// TIA Portal project "04_Kommisionierung_2018-10-11" (V14)
// Automatikbetribeb für das Modul "04-Kommisionierung" mit Factory IO

(* hardware
DEVICE "S7300/ET200M-Station_4"  S7-300 station
   slot 0: "Profilschiene_0"  Rail  6ES7 390-1***0-0AA0
   slot 1: "PS 307 5A_1"  PS 307 5A  6ES7 307-1EA01-0AA0
   slot 2: "PLC_Bus"  CPU 314C-2 DP  6ES7 314-6CH04-0AB0  V3.3
      slot 0: "MPI-Schnittstelle_1"  MPI
      slot 1: "DP-Schnittstelle_1"  DP
      slot 2: "DI 24/DO 16_1"  DI24/DO16
      slot 3: "AI 5/AO 2_1"  AI5/AO2
      slot 4: "Zählen_1"  Counter
      slot 5: "Positionieren_1"  Positioning
   slot 4: "DI 64x24VDC sinking/souring_1"  DI64 x 24VDC  6ES7 321-1BP00-0AA0
   slot 5: "DI 64x24VDC sinking/souring_2"  DI64 x 24VDC  6ES7 321-1BP00-0AA0
   slot 6: "DI 64x24VDC sinking/souring_3"  DI64 x 24VDC  6ES7 321-1BP00-0AA0
   slot 7: "DI 64x24VDC sinking/souring_4"  DI64 x 24VDC  6ES7 321-1BP00-0AA0
   slot 8: "DO 64x24VDC/0.3A sourcing_1"  DO64 x 24VDC / 0.3A, P  6ES7 322-1BP00-0AA0
   slot 9: "DO 64x24VDC/0.3A sourcing_2"  DO64 x 24VDC / 0.3A, P  6ES7 322-1BP00-0AA0
   slot 10: "DO 64x24VDC/0.3A sourcing_3"  DO64 x 24VDC / 0.3A, P  6ES7 322-1BP00-0AA0
   slot 11: "DO 64x24VDC/0.3A sourcing_4"  DO64 x 24VDC / 0.3A, P  6ES7 322-1BP00-0AA0
*)

// ===== PLC "PLC_Bus"  CPU 314C-2 DP =====

VAR_GLOBAL   // PLC tag table "Betriebsart"
   "S0_HS" AT %E0.0 : Bool;   // Hauptschalter 0-Aus, 1-Ein
   "S1_Not_Halt" AT %E0.1 : Bool;   // Not-Halt NC
   "S2_START" AT %E0.2 : Bool;   // Taster START NO
   "S3_STOP" AT %E0.3 : Bool;   // Taster STOP NC
   "Res_E04" AT %E0.4 : Bool;
   "Res_E05" AT %E0.5 : Bool;
   "Res_E06" AT %E0.6 : Bool;
   "Res_E07" AT %E0.7 : Bool;
   "Res_E10" AT %E1.0 : Bool;
   "Res_E11" AT %E1.1 : Bool;
   "Res_E12" AT %E1.2 : Bool;
   "Res_E13" AT %E1.3 : Bool;
   "Res_E14" AT %E1.4 : Bool;
   "Res_E15" AT %E1.5 : Bool;
   "Res_E16" AT %E1.6 : Bool;
   "Factory_IO_RUN" AT %E1.7 : Bool;   // Rückmeldung Factory IO läuft
   "P1_MS_RT" AT %A1.0 : Bool;   // Meldesäule Rot
   "P2_MS_GE" AT %A0.1 : Bool;   // Meldesäule Gelb
   "P3_MS_GN" AT %A0.2 : Bool;   // Meldesäule Grün
   "P10_START" AT %A0.3 : Bool;   // Anzeige grün in START-Taster
   "P11_STOP" AT %A0.4 : Bool;   // Anzeige gelb in STOP-Taster
   "Res_A0.5" AT %A0.5 : Bool;
   "P12_Anfahrwarnung" AT %A0.6 : Bool;   // Rundumleuchte System
   "P13_Sirene" AT %A0.7 : Bool;   // Sirene System
   "Res_A10" AT %A1.0 : Bool;
   "Res_A11" AT %A1.1 : Bool;
   "Res_A12" AT %A1.2 : Bool;
   "Res_A13" AT %A1.3 : Bool;
   "Res_A14" AT %A1.4 : Bool;
   "Res_A15" AT %A1.5 : Bool;
   "Res_A16" AT %A1.6 : Bool;
   "Res_A17" AT %A1.7 : Bool;
   "Log_1" AT %M0.1 : Bool;   // statisch "1"
   "Log_0" AT %M0.0 : Bool;   // statisch "0"
   "Takt_1HZ" AT %M100.5 : Bool;   // Taktmerker 1 Hz
END_VAR

VAR_GLOBAL   // PLC tag table "Kommisionierung"
   "B5001_TB5001" AT %E10.0 : Bool;   // Teil vom Emiiter vorhanden
   "B5002_TB5001" AT %E10.1 : Bool;   // Transportband-Ende
   "B5003_TB5002" AT %E10.2 : Bool;   // Transportband-Anfang
   "B5004_TB5002" AT %E10.3 : Bool;   // Transportband-Ende
   "B5005_TB5003" AT %E10.4 : Bool;   // Transportband-Anfang
   "B5006_TB5003" AT %E10.5 : Bool;   // Transportband-Ende
   "B5007_TB5004" AT %E10.6 : Bool;   // Transportband-Anfang
   "B5008_TB5004" AT %E10.7 : Bool;   // Transportband-Ende
   "B5009_TB5005" AT %E11.0 : Bool;   // Transportband-Anfang
   "B5010_TB5005" AT %E11.1 : Bool;   // Transportband-Ende
   "B5011_Farbteil_BL" AT %E11.2 : Bool;   // Farberkennung BL
   "B5012_Farbteil_GN" AT %E11.3 : Bool;   // Farberkennung GN
   "B5013_TB5006" AT %E11.4 : Bool;   // Transportband-Anfang
   "B5014_TB5006" AT %E11.5 : Bool;   // Transportband-Ende
   "B5015_Teil_in_Pos" AT %E11.6 : Bool;   // Teil in Abholposition
   "B5016_Teil_vorhanden" AT %E11.7 : Bool;   // Teil vom Emitter generiert
   "B5017_Teil_in_Pos" AT %E12.0 : Bool;   // Teil in Abholposition
   "B5018_Teil_vorhanden" AT %E12.1 : Bool;   // Teil vom Emitter generiert
   "B5019_TB5009" AT %E12.2 : Bool;   // Transportband-Anfang
   "B5020_TB5009" AT %E12.3 : Bool;   // Transportband-Ende
   "B5021_TB5010" AT %E12.4 : Bool;   // Transportband-Anfang
   "B5022_TB5010" AT %E12.5 : Bool;   // Transportband-Ende
   "Res_E126" AT %E12.6 : Bool;
   "Res_E127" AT %E12.7 : Bool;
   "B5030_PAP5001_RM_X" AT %E13.0 : Bool;
   "B5031_PAP5001_RM_Z" AT %E13.1 : Bool;
   "B5032_PAP5001_Teil_erkannt" AT %E13.2 : Bool;
   "B5040_PAP5002_RM_X" AT %E13.3 : Bool;
   "B5041_PAP5002_RM_Z" AT %E13.4 : Bool;
   "B5042_PAP5002_Teil_erkannt" AT %E13.5 : Bool;
   "Res_E136" AT %E13.6 : Bool;
   "Res_E137" AT %E13.7 : Bool;
   "TB5001" AT %A8.0 : Bool;
   "TB5002" AT %A8.1 : Bool;
   "TB5003" AT %A8.2 : Bool;
   "TB5004" AT %A8.3 : Bool;
   "TB5005" AT %A8.4 : Bool;
   "TB5006" AT %A8.5 : Bool;
   "TB5007" AT %A8.6 : Bool;
   "TB5008" AT %A8.7 : Bool;
   "TB5009" AT %A9.0 : Bool;
   "TB5010" AT %A9.1 : Bool;
   "STOP5001" AT %A9.2 : Bool;   // Stopper
   "STOP5002" AT %A9.3 : Bool;   // Stopper
   "STOP5003" AT %A9.4 : Bool;   // Stopper
   "STOP5004" AT %A9.5 : Bool;   // Stopper
   "STOP5005" AT %A9.6 : Bool;   // Stopper
   "Res_A97" AT %A9.7 : Bool;
   "PAP5001_X" AT %A10.0 : Bool;
   "PAP5001_Z" AT %A10.1 : Bool;
   "PAP5001_Greifer" AT %A10.2 : Bool;
   "PAP5002_X" AT %A10.3 : Bool;
   "PAP5002_Z" AT %A10.4 : Bool;
   "PAP5002_Greifer" AT %A10.5 : Bool;
   "Res_A106" AT %A10.6 : Bool;
   "Res_A107" AT %A10.7 : Bool;
   "RS5001_V" AT %A11.0 : Bool;   // Rollensorter Antrieb ein
   "RS5001_links" AT %A11.1 : Bool;   // Rollensorter Steuerung links
   "RS5001_rechts" AT %A11.2 : Bool;   // Rollensorter Steuerung rechts
   "Res_A113" AT %A11.3 : Bool;
   "Res_A114" AT %A11.4 : Bool;
   "Emitter_1" AT %A11.5 : Bool;
   "Emitter_2" AT %A11.6 : Bool;
   "Emitter_3" AT %A11.7 : Bool;
END_VAR

VAR_GLOBAL   // PLC tag table "KW_Variablen"
   "M_True" AT %M20.0 : Bool;   // Merker, der immer TRUE ist
   "M_False" AT %M20.1 : Bool;   // Merker, der immer FALSE ist
   "M_Beladen_Fern" AT %M22.0 : Bool;   // Merker, das Signal die ferne Ladestation zu aktivieren
   "M_Beladen_Nah" AT %M22.1 : Bool;   // Merker, das Signal die nähe Ladestation zu aktivieren
   "M_Abfuhr_Fern" AT %M22.2 : Bool;   // Merker, das Signal, dass das laden bei der fernen Ladestation beendet ist
   "M_Abfuhr_Nah" AT %M22.3 : Bool;   // Merker, das Signal, dass das laden bei der nähren Ladestation beendet ist
   "M_FRG_N1" AT %M22.4 : Bool;   // Merker, Freigabe Nummer 1
   "M_BND2_KB" AT %M22.5 : Bool;   // Merker Kiste beladen für das zweite Band
   "M_BND3_KB" AT %M22.6 : Bool;   // Merker Kiste beladen für das dritte Band
   "M_BND4_KB" AT %M22.7 : Bool;   // Merker Kiste beladen für das vierte Band
   "M_FRG_N2" AT %M23.0 : Bool;   // Merker, Freigabe Nummer 2
END_VAR

DATA_BLOCK "04-01 LoadLine_DB"   // DB1
{ S7_Optimized_Access := 'FALSE' }
VERSION : 0.1
// stored: InstanceOfName 04-01 LoadLine
"04-01 LoadLine"
BEGIN
END_DATA_BLOCK

DATA_BLOCK "04_00 Kistenerzeugung_DB"   // DB2
{ S7_Optimized_Access := 'FALSE' }
VERSION : 0.1
// stored: InstanceOfName 04-00 Kistenerzeugung
"04-00 Kistenerzeugung"
BEGIN
END_DATA_BLOCK

DATA_BLOCK "04-04 Sortierstation_DB"   // DB3
{ S7_Optimized_Access := 'FALSE' }
VERSION : 0.1
// stored: InstanceOfName 04-05 Sortierstation
"04-05 Sortierstation"
BEGIN
END_DATA_BLOCK

DATA_BLOCK "Kistengedaechnis_DB"   // DB4
{ S7_Optimized_Access := 'FALSE' }
VERSION : 0.1
// stored: InstanceOfName 04-02 Kistengedaechnis
"04-02 Kistengedaechnis"
BEGIN
END_DATA_BLOCK

DATA_BLOCK "PnP_Rueckw_01_DB"   // DB5
{ S7_Optimized_Access := 'FALSE' }
VERSION : 0.1
// stored: InstanceOfName Pick_n_Place_Rueckw
"Pick_n_Place_Rueckw"
BEGIN
END_DATA_BLOCK

DATA_BLOCK "PnP_Rueckw_02_DB"   // DB6
{ S7_Optimized_Access := 'FALSE' }
VERSION : 0.1
// stored: InstanceOfName Pick_n_Place_Rueckw
"Pick_n_Place_Rueckw"
BEGIN
END_DATA_BLOCK

DATA_BLOCK "FB_NC-NC_01_DB"   // DB7
{ S7_Optimized_Access := 'FALSE' }
VERSION : 0.1
// stored: InstanceOfName Foerderband_NC-NC
"Foerderband_NC-NC"
BEGIN
END_DATA_BLOCK

DATA_BLOCK "FB_NC-NC_02_DB"   // DB8
{ S7_Optimized_Access := 'FALSE' }
VERSION : 0.1
// stored: InstanceOfName Foerderband_NC-NC
"Foerderband_NC-NC"
BEGIN
END_DATA_BLOCK

DATA_BLOCK "FB_NC-NC_03_DB"   // DB9
{ S7_Optimized_Access := 'FALSE' }
VERSION : 0.1
// stored: InstanceOfName Foerderband_NC-NC
"Foerderband_NC-NC"
BEGIN
END_DATA_BLOCK

DATA_BLOCK "FB_NC-NC_04_DB"   // DB10
{ S7_Optimized_Access := 'FALSE' }
VERSION : 0.1
// stored: InstanceOfName Foerderband_NC-NC
"Foerderband_NC-NC"
BEGIN
END_DATA_BLOCK

FUNCTION_BLOCK "04-01 LoadLine"   // FB1, LAD
TITLE = Die lange gerade Fertigungslinie, wo die leere Kisten mit grünen und Blauen Teilen beladen werden
{ S7_Optimized_Access := 'FALSE' }
VERSION : 0.1
// Es darf gleichzeitig nur eine Kiste auf einem Band stehen, die ganze Logik der Programm geht davon aus, falls es mehr werden - gibt es Probleme, hier sind keine Mechamismen implementiert, die das erkennen. !!!Verbesserungsmöglichkeit!!!
   VAR_INPUT
      MTP_Sperre : Bool;   // Signal um den Motor SOFORT AUSzuschalten
      FRG_IN : Bool;   // Eingehende Freigabe vom nächsten Kettenglied
      BLDN_Fern : Bool;   // Signal, der auffordert die ferne Station die Kiste zum Laden zu stoppen
      BLDN_Nah : Bool;   // Signal, der auffordert die nähre Station die Kiste zum Laden zu stoppen
      ABFUHR_Fern : Bool;   // das laden ist beendet. die Kiste darf weiter fahren
      ABFUHR_Nah : Bool;   // das laden ist beendet. die Kiste darf weiter fahren
   END_VAR
   VAR_OUTPUT
      FRG_OUT : Bool;   // Freigabe für das vorherige Kettenglied
   END_VAR
   VAR
      TB_GNRL_01_DB : "TB_General";   // Instansdatenbaustein
      TB_GNRL_02_DB : "TB_General";   // Instansdatenbaustein
      TB_GNRL_03_DB : "TB_General";   // Instansdatenbaustein
      TB_GNRL_04_DB : "TB_General";   // Instansdatenbaustein
      FRG_VAL_1 : Bool;   // Freigabe-Signal für erste Band-Übergang (zwischen Bändern)
      FRG_VAL_2 : Bool;   // Freigabe-Signal für erste Band-Übergang (zwischen Bändern)
      FRG_VAL_3 : Bool;   // Freigabe-Signal für erste Band-Übergang (zwischen Bändern)
      STOP_1 : Bool;   // Aufforderung die Kiste in Lageposition zu stoppen, um zu beladen
      STOP_2 : Bool;   // Aufforderung die Kiste in Lageposition zu stoppen, um zu beladen
      Abfuhr_Modus_1 : Bool;   // Fordert auf die beladene Kiste weiterzuführen
      Abfuhr_Modus_2 : Bool;   // Fordert auf die beladene Kiste weiterzuführen
      flk_snsr_1 : Bool;   // flankenerkennunsbit
      flk_snsr_2 : Bool;   // flankenerkennunsbit
      FRG_OUT_Temp : Bool;   // Provisorische Variable
      Uebergabe_1 : Bool;   // Prüfen ob nütztlich, fall nicht - entfernen
      Uebergabe_2 : Bool;   // Prüfen ob nütztlich, fall nicht - entfernen
      flk_Abfuhr_Nah : Bool;   // flankenerkennunsbit
      flk_Abfuhr_Fern : Bool;   // flankenerkennunsbit
   END_VAR
   VAR_TEMP   // added for the SCL form of the ladder/FBD networks
      _w1 : Bool;
      _w2 : Bool;
   END_VAR
BEGIN

REGION Network 1: Erstes Band (1st LD-St)
   // Standardbeschaltung, Übergabe-Signal wird nicht benutzt, prüfen ob überhaupt nötig ist.
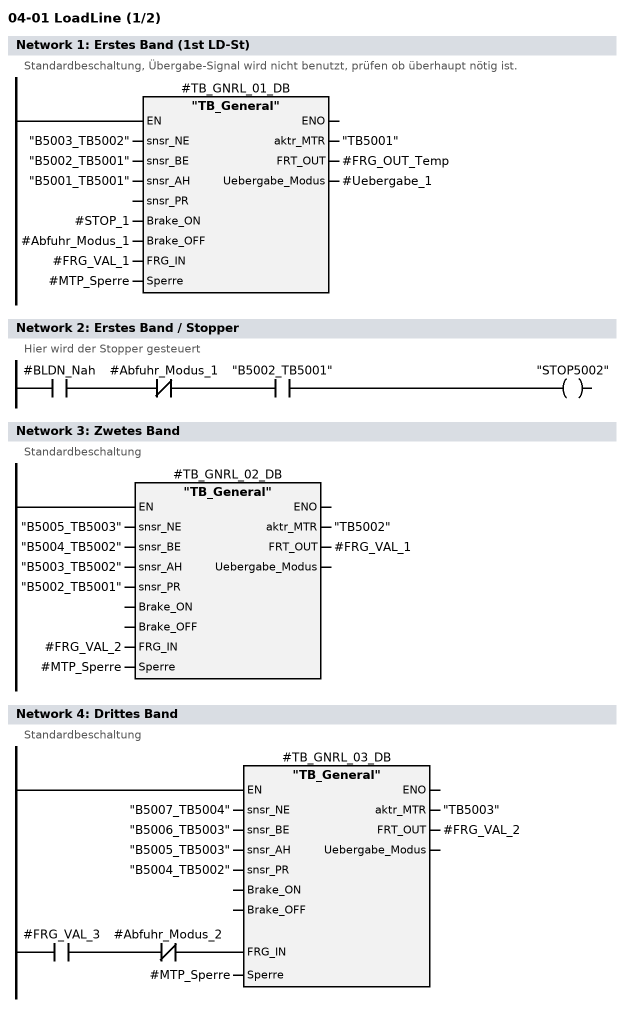
   RUNG wire#powerrail
      #TB_GNRL_01_DB(snsr_NE := "B5003_TB5002", snsr_BE := "B5002_TB5001", snsr_AH := "B5001_TB5001", snsr_PR :=, Brake_ON := #STOP_1, Brake_OFF := #Abfuhr_Modus_1, FRG_IN := #FRG_VAL_1, Sperre := #MTP_Sperre, aktr_MTR => "TB5001", FRT_OUT => #FRG_OUT_Temp, Uebergabe_Modus => #Uebergabe_1)
   END_RUNG
   // the same network as SCL:
   #TB_GNRL_01_DB(snsr_NE := "B5003_TB5002",   // "TB_General"
                  snsr_BE := "B5002_TB5001",
                  snsr_AH := "B5001_TB5001",
                  Brake_ON := #STOP_1,
                  Brake_OFF := #Abfuhr_Modus_1,
                  FRG_IN := #FRG_VAL_1,
                  Sperre := #MTP_Sperre,
                  aktr_MTR => "TB5001",
                  FRT_OUT => #FRG_OUT_Temp,
                  Uebergabe_Modus => #Uebergabe_1);
END_REGION

REGION Network 2: Erstes Band / Stopper
   // Hier wird der Stopper gesteuert
   RUNG wire#powerrail
      Contact( #BLDN_Nah )
      I_Contact( #Abfuhr_Modus_1 )
      Contact( "B5002_TB5001" )
      Coil( "STOP5002" )
   END_RUNG
   // the same network as SCL:
   "STOP5002" := #BLDN_Nah AND NOT #Abfuhr_Modus_1 AND "B5002_TB5001";
END_REGION

REGION Network 3: Zwetes Band
   // Standardbeschaltung
   RUNG wire#powerrail
      #TB_GNRL_02_DB(snsr_NE := "B5005_TB5003", snsr_BE := "B5004_TB5002", snsr_AH := "B5003_TB5002", snsr_PR := "B5002_TB5001", Brake_ON :=, Brake_OFF :=, FRG_IN := #FRG_VAL_2, Sperre := #MTP_Sperre, aktr_MTR => "TB5002", FRT_OUT => #FRG_VAL_1, Uebergabe_Modus =>)
   END_RUNG
   // the same network as SCL:
   #TB_GNRL_02_DB(snsr_NE := "B5005_TB5003",   // "TB_General"
                  snsr_BE := "B5004_TB5002",
                  snsr_AH := "B5003_TB5002",
                  snsr_PR := "B5002_TB5001",
                  FRG_IN := #FRG_VAL_2,
                  Sperre := #MTP_Sperre,
                  aktr_MTR => "TB5002",
                  FRT_OUT => #FRG_VAL_1);
END_REGION

REGION Network 4: Drittes Band
   // Standardbeschaltung
   RUNG wire#powerrail
      #TB_GNRL_03_DB(FRG_IN := wire#w1, snsr_NE := "B5007_TB5004", snsr_BE := "B5006_TB5003", snsr_AH := "B5005_TB5003", snsr_PR := "B5004_TB5002", Brake_ON :=, Brake_OFF :=, Sperre := #MTP_Sperre, aktr_MTR => "TB5003", FRT_OUT => #FRG_VAL_2, Uebergabe_Modus =>)
   END_RUNG
   RUNG wire#powerrail
      Contact( #FRG_VAL_3 )
      I_Contact( #Abfuhr_Modus_2 )
   END_RUNG wire#w1
   // the same network as SCL:
   #TB_GNRL_03_DB(snsr_NE := "B5007_TB5004",   // "TB_General"
                  snsr_BE := "B5006_TB5003",
                  snsr_AH := "B5005_TB5003",
                  snsr_PR := "B5004_TB5002",
                  FRG_IN := #FRG_VAL_3 AND NOT #Abfuhr_Modus_2,
                  Sperre := #MTP_Sperre,
                  aktr_MTR => "TB5003",
                  FRT_OUT => #FRG_VAL_2);
END_REGION

REGION Network 5: Viertes Band (2nd LD-St)
   // Standardbeschaltung
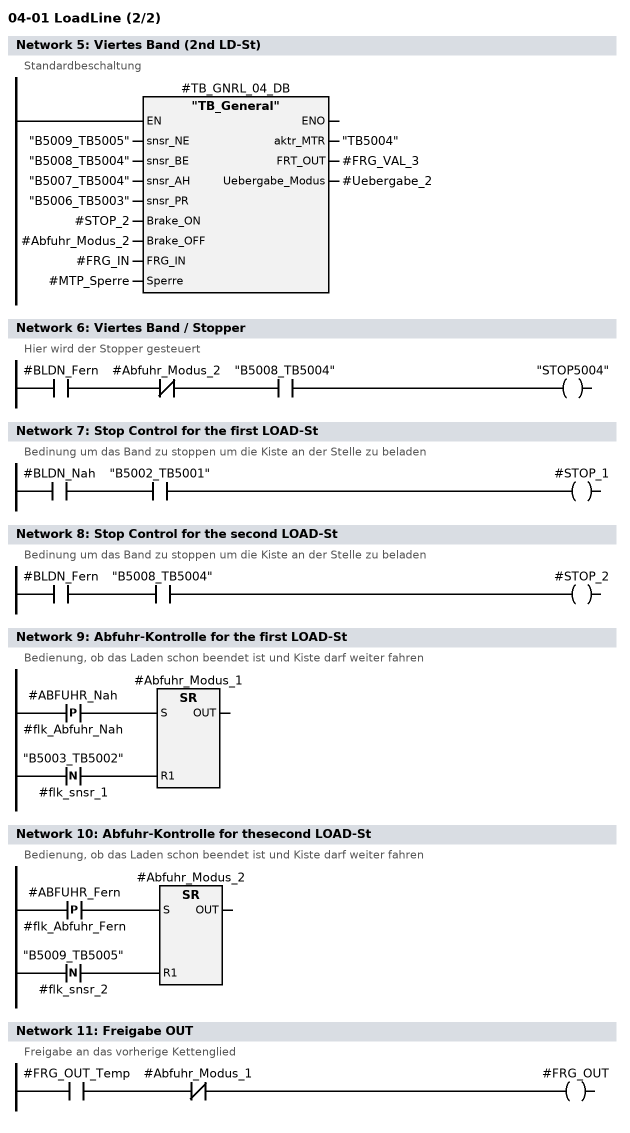
   RUNG wire#powerrail
      #TB_GNRL_04_DB(snsr_NE := "B5009_TB5005", snsr_BE := "B5008_TB5004", snsr_AH := "B5007_TB5004", snsr_PR := "B5006_TB5003", Brake_ON := #STOP_2, Brake_OFF := #Abfuhr_Modus_2, FRG_IN := #FRG_IN, Sperre := #MTP_Sperre, aktr_MTR => "TB5004", FRT_OUT => #FRG_VAL_3, Uebergabe_Modus => #Uebergabe_2)
   END_RUNG
   // the same network as SCL:
   #TB_GNRL_04_DB(snsr_NE := "B5009_TB5005",   // "TB_General"
                  snsr_BE := "B5008_TB5004",
                  snsr_AH := "B5007_TB5004",
                  snsr_PR := "B5006_TB5003",
                  Brake_ON := #STOP_2,
                  Brake_OFF := #Abfuhr_Modus_2,
                  FRG_IN := #FRG_IN,
                  Sperre := #MTP_Sperre,
                  aktr_MTR => "TB5004",
                  FRT_OUT => #FRG_VAL_3,
                  Uebergabe_Modus => #Uebergabe_2);
END_REGION

REGION Network 6: Viertes Band / Stopper
   // Hier wird der Stopper gesteuert
   RUNG wire#powerrail
      Contact( #BLDN_Fern )
      I_Contact( #Abfuhr_Modus_2 )
      Contact( "B5008_TB5004" )
      Coil( "STOP5004" )
   END_RUNG
   // the same network as SCL:
   "STOP5004" := #BLDN_Fern AND NOT #Abfuhr_Modus_2 AND "B5008_TB5004";
END_REGION

REGION Network 7: Stop Control for the first LOAD-St
   // Bedinung um das Band zu stoppen um die Kiste an der Stelle zu beladen
   RUNG wire#powerrail
      Contact( #BLDN_Nah )
      Contact( "B5002_TB5001" )
      Coil( #STOP_1 )
   END_RUNG
   // the same network as SCL:
   #STOP_1 := #BLDN_Nah AND "B5002_TB5001";
END_REGION

REGION Network 8: Stop Control for the second LOAD-St
   // Bedinung um das Band zu stoppen um die Kiste an der Stelle zu beladen
   RUNG wire#powerrail
      Contact( #BLDN_Fern )
      Contact( "B5008_TB5004" )
      Coil( #STOP_2 )
   END_RUNG
   // the same network as SCL:
   #STOP_2 := #BLDN_Fern AND "B5008_TB5004";
END_REGION

REGION Network 9: Abfuhr-Kontrolle for the first LOAD-St
   // Bedienung, ob das Laden schon beendet ist und Kiste darf weiter fahren
   RUNG wire#powerrail
      P_Contact(operand := #ABFUHR_Nah, bit := #flk_Abfuhr_Nah)
      S_SR(operand := #Abfuhr_Modus_1, r1 := wire#w1)
   END_RUNG
   RUNG wire#powerrail
      N_Contact(operand := "B5003_TB5002", bit := #flk_snsr_1)
   END_RUNG wire#w1
   // the same network as SCL:
   #_w1 := #ABFUHR_Nah AND NOT #flk_Abfuhr_Nah;   // rising edge of #ABFUHR_Nah
   #flk_Abfuhr_Nah := #ABFUHR_Nah;
   #_w2 := NOT "B5003_TB5002" AND #flk_snsr_1;   // falling edge of "B5003_TB5002"
   #flk_snsr_1 := "B5003_TB5002";
   IF #_w1 THEN
       #Abfuhr_Modus_1 := TRUE;   // SR flip-flop
   END_IF;
   IF #_w2 THEN #Abfuhr_Modus_1 := FALSE; END_IF;
END_REGION

REGION Network 10: Abfuhr-Kontrolle for thesecond LOAD-St
   // Bedienung, ob das Laden schon beendet ist und Kiste darf weiter fahren
   RUNG wire#powerrail
      P_Contact(operand := #ABFUHR_Fern, bit := #flk_Abfuhr_Fern)
      S_SR(operand := #Abfuhr_Modus_2, r1 := wire#w1)
   END_RUNG
   RUNG wire#powerrail
      N_Contact(operand := "B5009_TB5005", bit := #flk_snsr_2)
   END_RUNG wire#w1
   // the same network as SCL:
   #_w1 := #ABFUHR_Fern AND NOT #flk_Abfuhr_Fern;   // rising edge of #ABFUHR_Fern
   #flk_Abfuhr_Fern := #ABFUHR_Fern;
   #_w2 := NOT "B5009_TB5005" AND #flk_snsr_2;   // falling edge of "B5009_TB5005"
   #flk_snsr_2 := "B5009_TB5005";
   IF #_w1 THEN
       #Abfuhr_Modus_2 := TRUE;   // SR flip-flop
   END_IF;
   IF #_w2 THEN #Abfuhr_Modus_2 := FALSE; END_IF;
END_REGION

REGION Network 11: Freigabe OUT
   // Freigabe an das vorherige Kettenglied
   RUNG wire#powerrail
      Contact( #FRG_OUT_Temp )
      I_Contact( #Abfuhr_Modus_1 )
      Coil( #FRG_OUT )
   END_RUNG
   // the same network as SCL:
   #FRG_OUT := #FRG_OUT_Temp AND NOT #Abfuhr_Modus_1;
END_REGION
END_FUNCTION_BLOCK

FUNCTION_BLOCK "04-05 Sortierstation"   // FB2, FBD
TITLE = Sortierstation nach der Farbe, besteht aus 4 Teilen
{ S7_Optimized_Access := 'FALSE' }
VERSION : 0.1
// Zur Station gehört das Band vor der Weiche mit Farbsensoren, die Weiche selbst und das Band nach der Weiche und noch 2 Bänder, die nach links von der Weiche führen.
   VAR_INPUT
      FRG_IN_L : Bool;   // Freigabe für die linke Abführbänder
      FRG_IN_G : Bool;   // Freigebe für das geradestehende Abfährband
      Sperre : Bool;   // Befehl dem Motor sofort auszuschalten
   END_VAR
   VAR_OUTPUT
      FRG_OUT : Bool;   // Freigabemeldung an das vorherige Kettenglied
   END_VAR
   VAR
      TB_General_01_DB : "TB_General";   // Instansdatenbaustein
      TB_General_02_DB : "TB_General";   // Instansdatenbaustein
      TB_General_03_DB : "TB_General";   // Instansdatenbaustein
      TB_General_04_DB : "TB_General";   // Instansdatenbaustein
      FRG_Left : Bool;   // Freigabe von der linken Linie
      FRG_Gerade : Bool;   // Freigabe von dem band, das gerade steht
      FRG_Left_Mitte : Bool;   // Freigebe zwischen beiden Bänder in der linken Linie
      FRG_OUT_Temp : Bool;   // Provisorische Variable
      flk_snsr : Bool;   // Flankenerkennungbit
      Eingegangen : Bool;   // Signal aus Flankenerkennung, dass das Band mit Farbsensoren betretten wurde
      Teil_G : Bool;   // Grünes Teil ist erkannt
      Teil_B : Bool;   // Blaues Teil ist erkannt
      flk_snsr_2 : Bool;   // Flankenerkennungbit
      flk_snsr_3 : Bool;   // Flankenerkennungbit
      flk_snsr_4 : Bool;   // Flankenerkennungbit
      Band_FRGB : Bool;   // aktiv, wenn NUR eine Farbe aus 2 erkannt wirde
      flk_erkenn_l : Bool;   // Signal aus Flankenerkennung
      flk_erkenn_g : Bool;   // Signal aus Flankenerkennung
   END_VAR
   VAR_TEMP   // added for the SCL form of the ladder/FBD networks
      _w1 : Bool;
   END_VAR
BEGIN

REGION Network 1: fuenftes Band mit Farbsensoren
   // Hier ist noch Optimierungspotenzial da, was die eingehende Freigabe für das Band angeht, jetzt das Band darf das nächste Ladestück aufnehmen, sobald die beide nach der Weiche stehende Bänder auch leer sind, eigentlich das sollte nach Freilassung der Weiche schon sein.
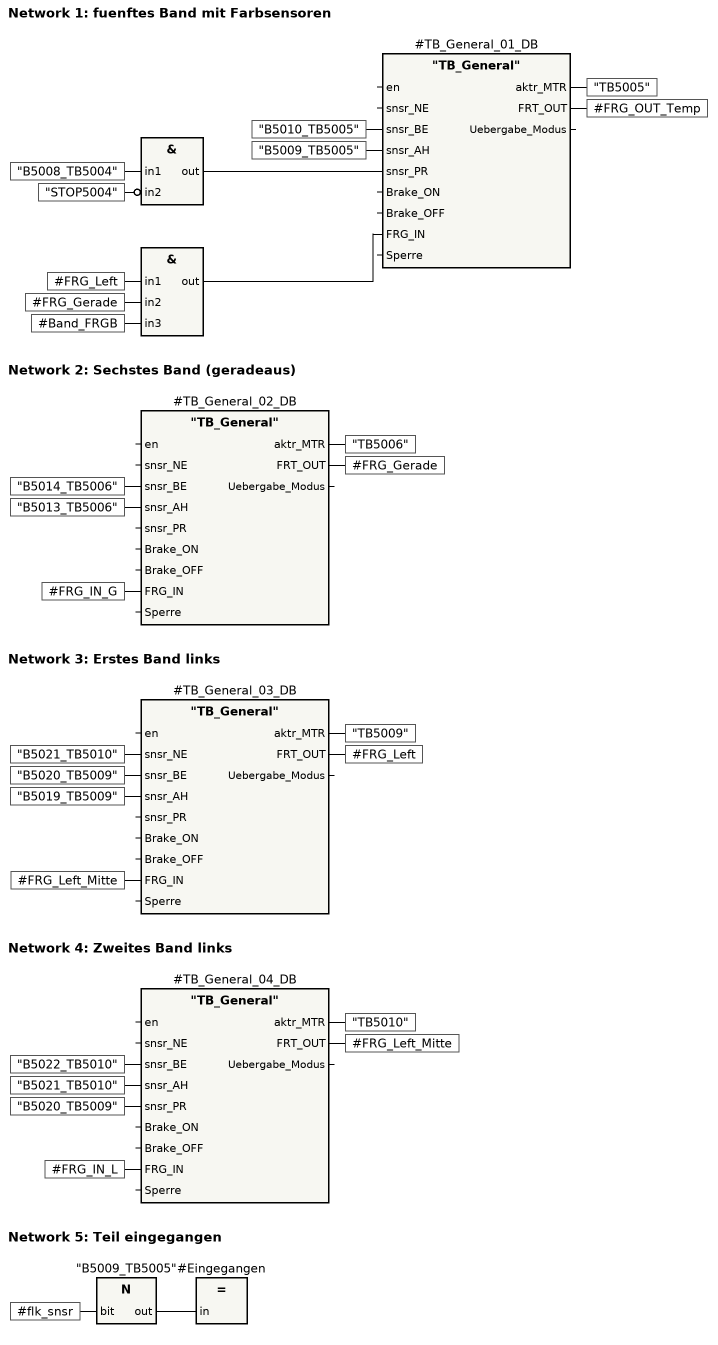
   #TB_General_01_DB(snsr_BE := "B5010_TB5005",   // "TB_General"
                     snsr_AH := "B5009_TB5005",
                     snsr_PR := "B5008_TB5004" AND NOT "STOP5004",
                     FRG_IN := #FRG_Left AND #FRG_Gerade AND #Band_FRGB,
                     aktr_MTR => "TB5005",
                     FRT_OUT => #FRG_OUT_Temp);
END_REGION

REGION Network 2: Sechstes Band (geradeaus)
   // Standardbeschaltung
   #TB_General_02_DB(snsr_BE := "B5014_TB5006",   // "TB_General"
                     snsr_AH := "B5013_TB5006",
                     FRG_IN := #FRG_IN_G,
                     aktr_MTR => "TB5006",
                     FRT_OUT => #FRG_Gerade);
END_REGION

REGION Network 3: Erstes Band links
   // Standardbeschaltung
   #TB_General_03_DB(snsr_NE := "B5021_TB5010",   // "TB_General"
                     snsr_BE := "B5020_TB5009",
                     snsr_AH := "B5019_TB5009",
                     FRG_IN := #FRG_Left_Mitte,
                     aktr_MTR => "TB5009",
                     FRT_OUT => #FRG_Left);
END_REGION

REGION Network 4: Zweites Band links
   // Standardbeschaltung
   #TB_General_04_DB(snsr_BE := "B5022_TB5010",   // "TB_General"
                     snsr_AH := "B5021_TB5010",
                     snsr_PR := "B5020_TB5009",
                     FRG_IN := #FRG_IN_L,
                     aktr_MTR => "TB5010",
                     FRT_OUT => #FRG_Left_Mitte);
END_REGION

REGION Network 5: Teil eingegangen
   // ist =1 für ein Zyklus
   #_w1 := NOT "B5009_TB5005" AND #flk_snsr;   // falling edge of "B5009_TB5005"
   #flk_snsr := "B5009_TB5005";
   #Eingegangen := #_w1;
END_REGION

REGION Network 6: Grün erkannt
   // Flip-Flop, wird gesetzt wenn die grüne Farbe erkannt wurde
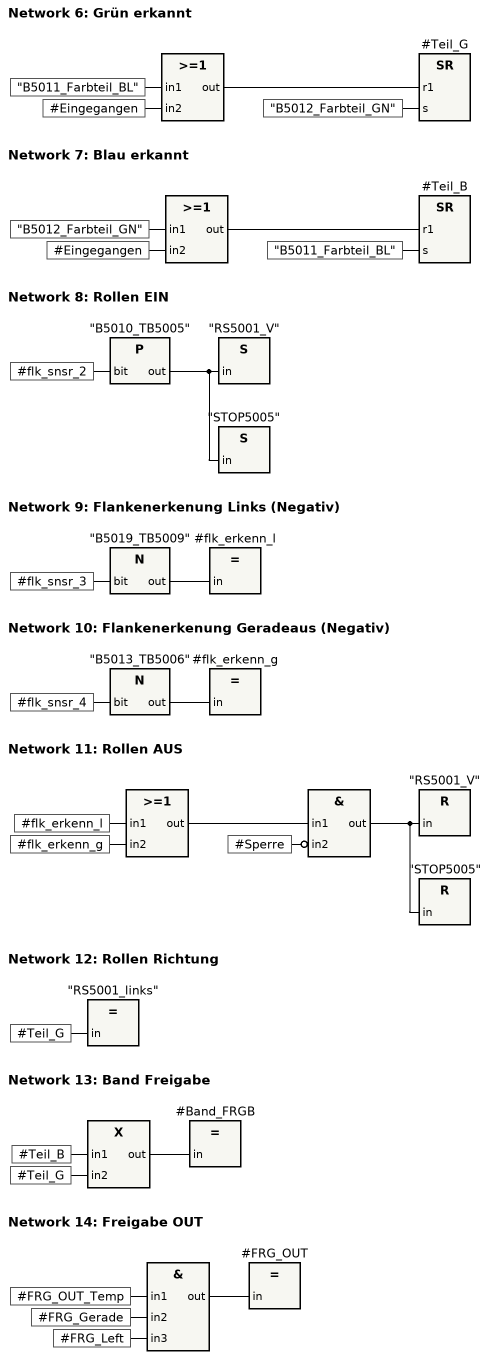
   IF "B5012_Farbteil_GN" THEN
       #Teil_G := TRUE;   // SR flip-flop
   END_IF;
   IF "B5011_Farbteil_BL" OR #Eingegangen THEN #Teil_G := FALSE; END_IF;
END_REGION

REGION Network 7: Blau erkannt
   // Flip-Flop, wird gesetzt wenn die blaue Farbe erkannt wurde
   IF "B5011_Farbteil_BL" THEN
       #Teil_B := TRUE;   // SR flip-flop
   END_IF;
   IF "B5012_Farbteil_GN" OR #Eingegangen THEN #Teil_B := FALSE; END_IF;
END_REGION

REGION Network 8: Rollen EIN
   // Setzt die Rollen und der Stopper der Weiche
   #_w1 := "B5010_TB5005" AND NOT #flk_snsr_2;   // rising edge of "B5010_TB5005"
   #flk_snsr_2 := "B5010_TB5005";
   IF #_w1 THEN
       "RS5001_V" := TRUE;
       "STOP5005" := TRUE;
   END_IF;
END_REGION

REGION Network 9: Flankenerkenung Links (Negativ)
   // wird am meheren Stellen verwendet
   #_w1 := NOT "B5019_TB5009" AND #flk_snsr_3;   // falling edge of "B5019_TB5009"
   #flk_snsr_3 := "B5019_TB5009";
   #flk_erkenn_l := #_w1;
END_REGION

REGION Network 10: Flankenerkenung Geradeaus (Negativ)
   // wird am meheren Stellen verwendet
   #_w1 := NOT "B5013_TB5006" AND #flk_snsr_4;   // falling edge of "B5013_TB5006"
   #flk_snsr_4 := "B5013_TB5006";
   #flk_erkenn_g := #_w1;
END_REGION

REGION Network 11: Rollen AUS
   // Rücksetzt die Rollen und der Stopper der Weiche
   IF (#flk_erkenn_l OR #flk_erkenn_g) AND NOT #Sperre THEN
       "RS5001_V" := FALSE;
       "STOP5005" := FALSE;
   END_IF;
END_REGION

REGION Network 12: Rollen Richtung
   // Grüne nach Links, die Blaue - geradeaus
   "RS5001_links" := #Teil_G;
END_REGION

REGION Network 13: Band Freigabe
   // XOR sorgt dafür, dass es eine EINZIGE Farbe erkannt werden darf, sonst geht nicht mehr weiter.
   #Band_FRGB := #Teil_B XOR #Teil_G;
END_REGION

REGION Network 14: Freigabe OUT
   // Freibage für das vorherige Kettenglied
   #FRG_OUT := #FRG_OUT_Temp AND #FRG_Gerade AND #FRG_Left;
END_REGION
END_FUNCTION_BLOCK

FUNCTION_BLOCK "04-02 Kistengedaechnis"   // FB3, FBD
TITLE = Speichert den Vervendungszweck jeder Kiste zwischen beiden Ladestationen
{ S7_Optimized_Access := 'FALSE' }
VERSION : 0.1
// Es gibt 3 globale Merker für jedes Band, wo Kistenstatus gespeichert und weitergegeben wird
   VAR
      flk_snsr_1 : Bool;
      flk_snsr_2 : Bool;
      flk_snsr_3 : Bool;
      flk_snsr_4 : Bool;
      flk_snsr_5 : Bool;
      flk_snsr_6 : Bool;
   END_VAR
   VAR_TEMP   // added for the SCL form of the ladder/FBD networks
      _w1 : Bool;
      _w2 : Bool;
   END_VAR
BEGIN

REGION Network 1: Kiste beladen auf zweitem Band
   // Wenn Merker aktiv ist, dann bedeutet, dass die Kiste auf diesem Band schon beladen ist, andersrum - leer
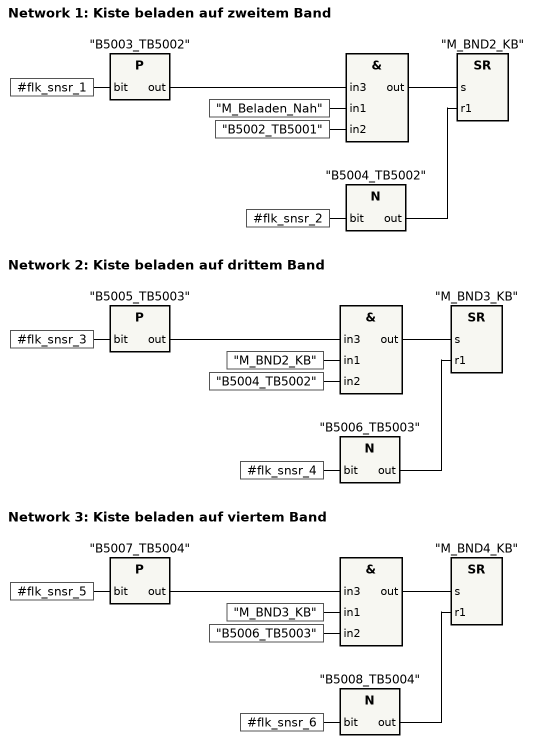
   #_w1 := "B5003_TB5002" AND NOT #flk_snsr_1;   // rising edge of "B5003_TB5002"
   #flk_snsr_1 := "B5003_TB5002";
   #_w2 := NOT "B5004_TB5002" AND #flk_snsr_2;   // falling edge of "B5004_TB5002"
   #flk_snsr_2 := "B5004_TB5002";
   IF #_w1 AND "M_Beladen_Nah" AND "B5002_TB5001" THEN
       "M_BND2_KB" := TRUE;   // SR flip-flop
   END_IF;
   IF #_w2 THEN "M_BND2_KB" := FALSE; END_IF;
END_REGION

REGION Network 2: Kiste beladen auf drittem Band
   // Wenn Merker aktiv ist, dann bedeutet, dass die Kiste auf diesem Band schon beladen ist, andersrum - leer
   #_w1 := "B5005_TB5003" AND NOT #flk_snsr_3;   // rising edge of "B5005_TB5003"
   #flk_snsr_3 := "B5005_TB5003";
   #_w2 := NOT "B5006_TB5003" AND #flk_snsr_4;   // falling edge of "B5006_TB5003"
   #flk_snsr_4 := "B5006_TB5003";
   IF #_w1 AND "M_BND2_KB" AND "B5004_TB5002" THEN
       "M_BND3_KB" := TRUE;   // SR flip-flop
   END_IF;
   IF #_w2 THEN "M_BND3_KB" := FALSE; END_IF;
END_REGION

REGION Network 3: Kiste beladen auf viertem Band
   // Wenn Merker aktiv ist, dann bedeutet, dass die Kiste auf diesem Band schon beladen ist, andersrum - leer
   #_w1 := "B5007_TB5004" AND NOT #flk_snsr_5;   // rising edge of "B5007_TB5004"
   #flk_snsr_5 := "B5007_TB5004";
   #_w2 := NOT "B5008_TB5004" AND #flk_snsr_6;   // falling edge of "B5008_TB5004"
   #flk_snsr_6 := "B5008_TB5004";
   IF #_w1 AND "M_BND3_KB" AND "B5006_TB5003" THEN
       "M_BND4_KB" := TRUE;   // SR flip-flop
   END_IF;
   IF #_w2 THEN "M_BND4_KB" := FALSE; END_IF;
END_REGION
END_FUNCTION_BLOCK

FUNCTION_BLOCK "04-00 Kistenerzeugung"   // FB4, FBD
TITLE = Kistenerzeugung von 2 Arten: NAH und FENR
{ S7_Optimized_Access := 'FALSE' }
VERSION : 0.1
// Die Kisten für beide Stationen werden immer abwechselnd erzeugt und dementsprechend markiert
   VAR_INPUT
      FRG_IN : Bool;   // eingehende Freigabe vom nächsten Kettenglied
      Start : Bool;   // Signal zum Starten
      snsr_V : Bool;   // Sensor vorne, wo die Kiste erzeugt wird
   END_VAR
   VAR_OUTPUT
      Emmiter : Bool;   // Ausgang, der direkt Kistenemmiter steuert
      Kiste_Nah : Bool;   // Kiste ist für nähere Ladestation markiert
      Kiste_Fern : Bool;   // Kiste ist für ferne Ladestation markiert
   END_VAR
   VAR
      flk_FRG_IN : Bool;   // Flankenerkennunsbit
      DoIt : Bool;   // wenn aktiv (=1) wird eine neue Kiste erzeugt
      flk_snsr_V : Bool;   // Flankenerkennunsbit
   END_VAR
   VAR_TEMP   // added for the SCL form of the ladder/FBD networks
      _w1 : Bool;
   END_VAR
BEGIN

REGION Network 1: Flanken Erkennung
   // Erkennung des Momentes wenn das Band freigeworden ist
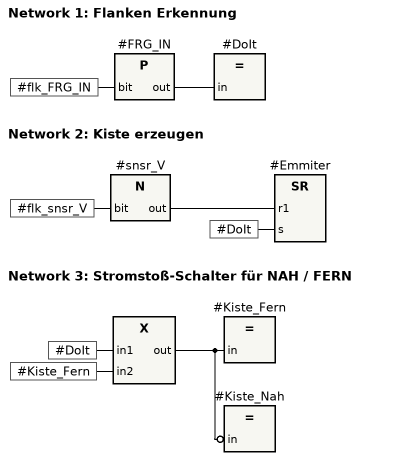
   #_w1 := #FRG_IN AND NOT #flk_FRG_IN;   // rising edge of #FRG_IN
   #flk_FRG_IN := #FRG_IN;
   #DoIt := #_w1;
END_REGION

REGION Network 2: Kiste erzeugen
   // Der Emmitter in Factory IO funkzioniert nicht immer vernünftig mit Aktivirung durch ein einziger Takt, deswegen Verzögerung
   #_w1 := NOT #snsr_V AND #flk_snsr_V;   // falling edge of #snsr_V
   #flk_snsr_V := #snsr_V;
   IF #DoIt THEN
       #Emmiter := TRUE;   // SR flip-flop
   END_IF;
   IF #_w1 THEN #Emmiter := FALSE; END_IF;
END_REGION

REGION Network 3: Stromstoß-Schalter für NAH / FERN
   // Wird abwächseld nahe  und ferne Kiste hergestellt
   #Kiste_Fern := #DoIt XOR #Kiste_Fern;
   #Kiste_Nah := NOT #Kiste_Fern;
END_REGION
END_FUNCTION_BLOCK

FUNCTION_BLOCK "Foerderband_NC-NC"   // FB5, LAD
TITLE = Einfache Steuerung für das Förderband mit Öffner-Sensoren (Lichtschranke mit dem Spigel)
{ S7_Optimized_Access := 'FALSE' }
VERSION : 0.1
// Wurde als Grundlage aus einem früherem Project übernommen, kann grundsätztlich durch TB_General ersetzt werden (erstmal prüfen!)
   VAR_INPUT
      Erster_Sensor : Bool;   // Der erste sensor der Ladung überwacht in Laufrichtung (NC)
      Letzter_Sensor : Bool;   // Der zweite sensor der Ladung überwacht in Laufrichtung (NC)
      Freigabe : Bool;   // Freigabe-Signal von nächstem Kettenglied (Station oder Band)
      Motor_AN : Bool;   // Aufforderung Motor ANzuschalten, solange Signal aktiv ist
      Sperre : Bool;   // Befehl den Motor sofort AUSzuschalten
   END_VAR
   VAR_OUTPUT
      Motor : Bool;   // Ausgang, der den Motor steuert aktiv =1
      Bereit : Bool;   // Bereitschaf an das vorherige Kettenglied zu melden
   END_VAR
   VAR
      Beladen : Bool;   // Das Band ist mit Ladestück beladen
      FLK_ErsterSensor : Bool;   // Flankenerkennunsbit
      FLK_LetzterSensor : Bool;   // Flankenerkennunsbit
   END_VAR
   VAR_TEMP   // added for the SCL form of the ladder/FBD networks
      _w1 : Bool;
   END_VAR
BEGIN

REGION Network 1: Beladen wird EIN
   // Sobald der erster Sensor (Lichtschranke) betätigt ist, gilt die Förderbahn als mit der Last (Teil) beladen.
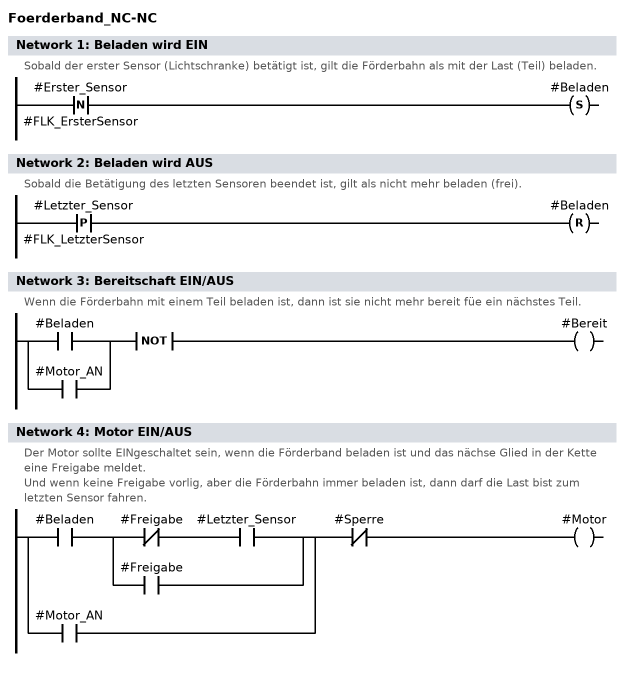
   RUNG wire#powerrail
      N_Contact(operand := #Erster_Sensor, bit := #FLK_ErsterSensor)
      S_Coil( #Beladen )
   END_RUNG
   // the same network as SCL:
   #_w1 := NOT #Erster_Sensor AND #FLK_ErsterSensor;   // falling edge of #Erster_Sensor
   #FLK_ErsterSensor := #Erster_Sensor;
   IF #_w1 THEN #Beladen := TRUE; END_IF;
END_REGION

REGION Network 2: Beladen wird AUS
   // Sobald die Betätigung des letzten Sensoren beendet ist, gilt als nicht mehr beladen (frei).
   RUNG wire#powerrail
      P_Contact(operand := #Letzter_Sensor, bit := #FLK_LetzterSensor)
      R_Coil( #Beladen )
   END_RUNG
   // the same network as SCL:
   #_w1 := #Letzter_Sensor AND NOT #FLK_LetzterSensor;   // rising edge of #Letzter_Sensor
   #FLK_LetzterSensor := #Letzter_Sensor;
   IF #_w1 THEN #Beladen := FALSE; END_IF;
END_REGION

REGION Network 3: Bereitschaft EIN/AUS
   // Wenn die Förderbahn mit einem Teil beladen ist, dann ist sie nicht mehr bereit füe ein nächstes Teil.
   RUNG wire#powerrail
      Contact( #Beladen )
      wire#w1
      Not()
      Coil( #Bereit )
   END_RUNG
   RUNG wire#powerrail
      Contact( #Motor_AN )
   END_RUNG wire#w1
   // the same network as SCL:
   #Bereit := NOT (#Beladen OR #Motor_AN);
END_REGION

REGION Network 4: Motor EIN/AUS
   // Der Motor sollte EINgeschaltet sein, wenn die Förderband beladen ist und das nächse Glied in der Kette eine Freigabe meldet. 
   // Und wenn keine Freigabe vorlig, aber die Förderbahn immer beladen ist, dann darf die Last bist zum letzten Sensor fahren.
   #Motor := ((#Beladen AND (#Freigabe OR (NOT #Freigabe AND #Letzter_Sensor))) OR #Motor_AN) AND NOT #Sperre;
END_REGION
END_FUNCTION_BLOCK

FUNCTION_BLOCK "TB_General"   // FB20, LAD
TITLE = Allgemeine Steuerung eines Foerderbandes
{ S7_Optimized_Access := 'FALSE' }
VERSION : 0.1
   VAR_INPUT
      snsr_NE : Bool;   // (NEXT) Erster Sensor beim nächsten Glied in der Kette
      snsr_BE : Bool;   // (BEHIND) Sensor hinten
      snsr_AH : Bool;   // (AHEAD) Sensor vorne
      snsr_PR : Bool;   // (PREVIOUS) Letzter Sensor beim vorherigen Kettenglied
      Brake_ON : Bool;   // Signal das Band zu stoppen
      Brake_OFF : Bool;   // Signal das Stoppen zurückzunehmen
      FRG_IN : Bool;   // Freigabe vom nächsten Kettenglied
      Sperre : Bool;   // Motorsperre, aktiv =1
   END_VAR
   VAR_OUTPUT
      aktr_MTR : Bool;   // Ausgang zum Steuern des Motores
      FRT_OUT : Bool;   // Freigabe zum vorherigen Kettenglied
      Uebergabe_Modus : Bool;   // Signal, dass Übergabemodus aktiv ist
   END_VAR
   VAR
      Loaded : Bool;   // Das Band ist beladen mit Ladestück
      Movement : Bool;   // Bedinung um Motror ANzuschalten
      Brake_Bypass : Bool;   // Bremsebefehl umzugehen
      flk_snsr_NE : Bool;   // flanken Erkennungsbit
      flk_snsr_BE_N : Bool;   // flanken Erkennungsbit
      flk_snsr_BE_P : Bool;   // flanken Erkennungsbit
      flk_snsr_AH : Bool;   // flanken Erkennungsbit
      flk_snsr_PR : Bool;   // flanken Erkennungsbit
      flk_Auswer_BE_N : Bool;   // Signal aus Flankenerkennung
      flk_Auswer_AH_P : Bool;   // Signal aus Flankenerkennung
      flk_Brake_OFF : Bool;   // flanken Erkennungsbit
   END_VAR
   VAR_TEMP   // added for the SCL form of the ladder/FBD networks
      _w1 : Bool;
   END_VAR
BEGIN

REGION Network 1: Flankenauswertung snsr_BE (Negativ)
   // Signal wird generiert, wenn das Ladestück den hinteren Sensor verlässt.
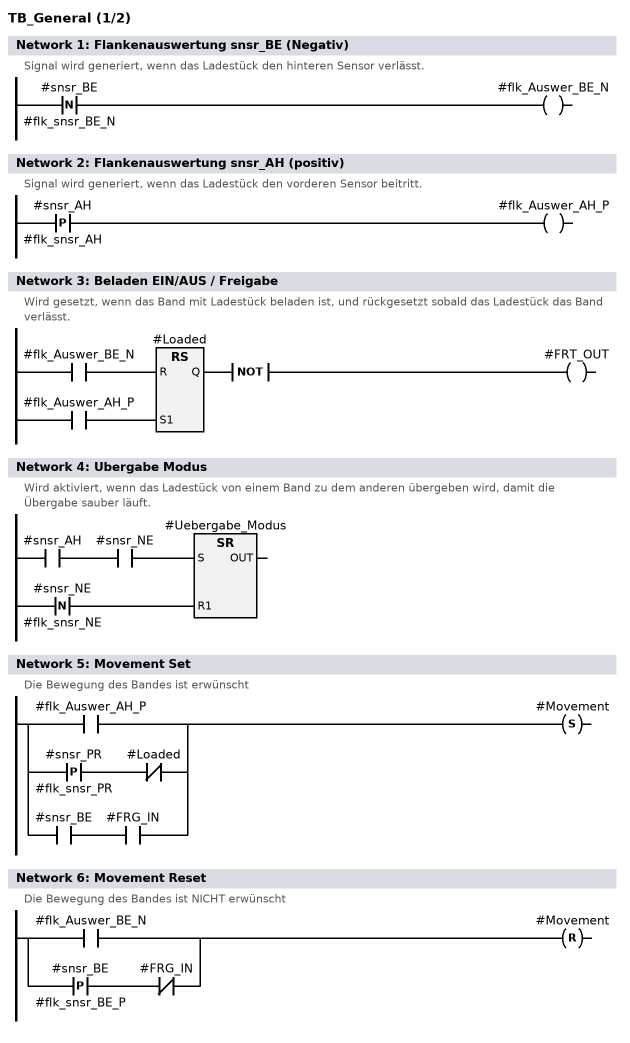
   RUNG wire#powerrail
      N_Contact(operand := #snsr_BE, bit := #flk_snsr_BE_N)
      Coil( #flk_Auswer_BE_N )
   END_RUNG
   // the same network as SCL:
   #_w1 := NOT #snsr_BE AND #flk_snsr_BE_N;   // falling edge of #snsr_BE
   #flk_snsr_BE_N := #snsr_BE;
   #flk_Auswer_BE_N := #_w1;
END_REGION

REGION Network 2: Flankenauswertung snsr_AH (positiv)
   // Signal wird generiert, wenn das Ladestück den vorderen Sensor beitritt.
   RUNG wire#powerrail
      P_Contact(operand := #snsr_AH, bit := #flk_snsr_AH)
      Coil( #flk_Auswer_AH_P )
   END_RUNG
   // the same network as SCL:
   #_w1 := #snsr_AH AND NOT #flk_snsr_AH;   // rising edge of #snsr_AH
   #flk_snsr_AH := #snsr_AH;
   #flk_Auswer_AH_P := #_w1;
END_REGION

REGION Network 3: Beladen EIN/AUS / Freigabe
   // Wird gesetzt, wenn das Band mit Ladestück beladen ist, und rückgesetzt sobald das Ladestück das Band verlässt.
   RUNG wire#powerrail
      Contact( #flk_Auswer_BE_N )
      S_RS(operand := #Loaded, s1 := wire#w1)
      Not()
      Coil( #FRT_OUT )
   END_RUNG
   RUNG wire#powerrail
      Contact( #flk_Auswer_AH_P )
   END_RUNG wire#w1
   // the same network as SCL:
   IF #flk_Auswer_BE_N THEN
       #Loaded := FALSE;   // RS flip-flop
   END_IF;
   IF #flk_Auswer_AH_P THEN #Loaded := TRUE; END_IF;
   #FRT_OUT := NOT #Loaded;
END_REGION

REGION Network 4: Ubergabe Modus
   // Wird aktiviert, wenn das Ladestück von einem Band zu dem anderen übergeben wird, damit die Übergabe sauber läuft.
   RUNG wire#powerrail
      Contact( #snsr_AH )
      Contact( #snsr_NE )
      S_SR(operand := #Uebergabe_Modus, r1 := wire#w1)
   END_RUNG
   RUNG wire#powerrail
      N_Contact(operand := #snsr_NE, bit := #flk_snsr_NE)
   END_RUNG wire#w1
   // the same network as SCL:
   #_w1 := NOT #snsr_NE AND #flk_snsr_NE;   // falling edge of #snsr_NE
   #flk_snsr_NE := #snsr_NE;
   IF #snsr_AH AND #snsr_NE THEN
       #Uebergabe_Modus := TRUE;   // SR flip-flop
   END_IF;
   IF #_w1 THEN #Uebergabe_Modus := FALSE; END_IF;
END_REGION

REGION Network 5: Movement Set
   // Die Bewegung des Bandes ist erwünscht
   RUNG wire#powerrail
      Contact( #flk_Auswer_AH_P )
      wire#w1
      S_Coil( #Movement )
   END_RUNG
   RUNG wire#powerrail
      P_Contact(operand := #snsr_PR, bit := #flk_snsr_PR)
      I_Contact( #Loaded )
   END_RUNG wire#w1
   RUNG wire#powerrail
      Contact( #snsr_BE )
      Contact( #FRG_IN )
   END_RUNG wire#w1
   // the same network as SCL:
   #_w1 := #snsr_PR AND NOT #flk_snsr_PR;   // rising edge of #snsr_PR
   #flk_snsr_PR := #snsr_PR;
   IF #flk_Auswer_AH_P OR (#_w1 AND NOT #Loaded) OR (#snsr_BE AND #FRG_IN) THEN #Movement := TRUE; END_IF;
END_REGION

REGION Network 6: Movement Reset
   // Die Bewegung des Bandes ist NICHT erwünscht
   RUNG wire#powerrail
      Contact( #flk_Auswer_BE_N )
      wire#w1
      R_Coil( #Movement )
   END_RUNG
   RUNG wire#powerrail
      P_Contact(operand := #snsr_BE, bit := #flk_snsr_BE_P)
      I_Contact( #FRG_IN )
   END_RUNG wire#w1
   // the same network as SCL:
   #_w1 := #snsr_BE AND NOT #flk_snsr_BE_P;   // rising edge of #snsr_BE
   #flk_snsr_BE_P := #snsr_BE;
   IF #flk_Auswer_BE_N OR (#_w1 AND NOT #FRG_IN) THEN #Movement := FALSE; END_IF;
END_REGION

REGION Network 7: Bremsenumgehung
   // Das Signal zum Anhalten wird damit überbrückt
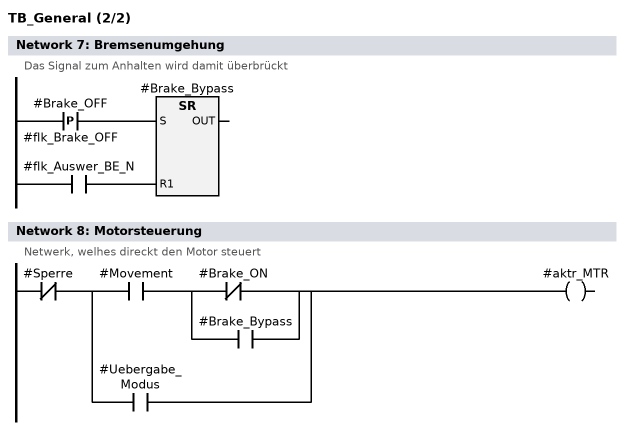
   RUNG wire#powerrail
      P_Contact(operand := #Brake_OFF, bit := #flk_Brake_OFF)
      S_SR(operand := #Brake_Bypass, r1 := wire#w1)
   END_RUNG
   RUNG wire#powerrail
      Contact( #flk_Auswer_BE_N )
   END_RUNG wire#w1
   // the same network as SCL:
   #_w1 := #Brake_OFF AND NOT #flk_Brake_OFF;   // rising edge of #Brake_OFF
   #flk_Brake_OFF := #Brake_OFF;
   IF #_w1 THEN
       #Brake_Bypass := TRUE;   // SR flip-flop
   END_IF;
   IF #flk_Auswer_BE_N THEN #Brake_Bypass := FALSE; END_IF;
END_REGION

REGION Network 8: Motorsteuerung
   // Netwerk, welhes direckt den Motor steuert
   RUNG wire#powerrail
      I_Contact( #Sperre )
      wire#w1
      Contact( #Movement )
      wire#w2
      I_Contact( #Brake_ON )
      wire#w3
      Coil( #aktr_MTR )
   END_RUNG
   RUNG wire#w2
      Contact( #Brake_Bypass )
   END_RUNG wire#w3
   RUNG wire#w1
      Contact( #Uebergabe_Modus )
   END_RUNG wire#w3
   // the same network as SCL:
   #aktr_MTR := NOT #Sperre AND ((#Movement AND (NOT #Brake_ON OR #Brake_Bypass)) OR #Uebergabe_Modus);
END_REGION
END_FUNCTION_BLOCK

FUNCTION_BLOCK "Pick_n_Place_Rueckw"   // FB95, LAD
TITLE = Ablaufkette für das Pick and Place Manipulator
{ S7_Optimized_Access := 'FALSE' }
VERSION : 0.1
// Nach Schrittkettenprinzip programmiert, aber Scritt Nummer 0 (Initialschritt) ist nicht optimal gelöst, die reinfolge der Netzwerke, die die Schritte darstellen solten lieber in ungekehrter Reinfolge, erstmal die Letze und dann die erste Schritte.
   VAR_INPUT
      snsr_X : Bool;
      snsr_Z : Bool;
      snsr_TE : Bool;
      snsr_HLN : Bool;
      snsr_ABLGN : Bool;
      "NOT-HALT" : Bool;
   END_VAR
   VAR_OUTPUT
      aktr_X : Bool;
      aktr_Z : Bool;
      aktr_GRFR : Bool;
      Uebernom : Bool;
      Freigelas : Bool;
      Fehler_NE : Bool;
   END_VAR
   VAR
      X0 : Bool;
      X1 : Bool;
      X2 : Bool;
      X3 : Bool;
      X4 : Bool;
      X5 : Bool;
      X6 : Bool;
      X7 : Bool;
      X8 : Bool;
      X9 : Bool;
      IF_X1 : Bool;
      IF_X2 : Bool;
      IF_X3 : Bool;
      IF_X4 : Bool;
      IF_X5 : Bool;
      IF_X6 : Bool;
      IF_X7 : Bool;
      IF_X8 : Bool;
      IF_X9 : Bool;
      flk_X1 : Bool;
      flk_X2 : Bool;
      flk_X3 : Bool;
      flk_X4 : Bool;
      flk_X5 : Bool;
      flk_X6 : Bool;
      flk_X7 : Bool;
      flk_X8 : Bool;
      flk_X9 : Bool;
      Zmove_ended : Bool;
      Xmove_ended : Bool;
      flk_Xmove : Bool;
      flk_Zmove : Bool;
      tmp_Flagge : Bool;
   END_VAR
   VAR_TEMP   // added for the SCL form of the ladder/FBD networks
      _w1 : Bool;
   END_VAR
BEGIN

REGION Network 1: Schritt 1/ Aus Grundstellung leer rueberfahren
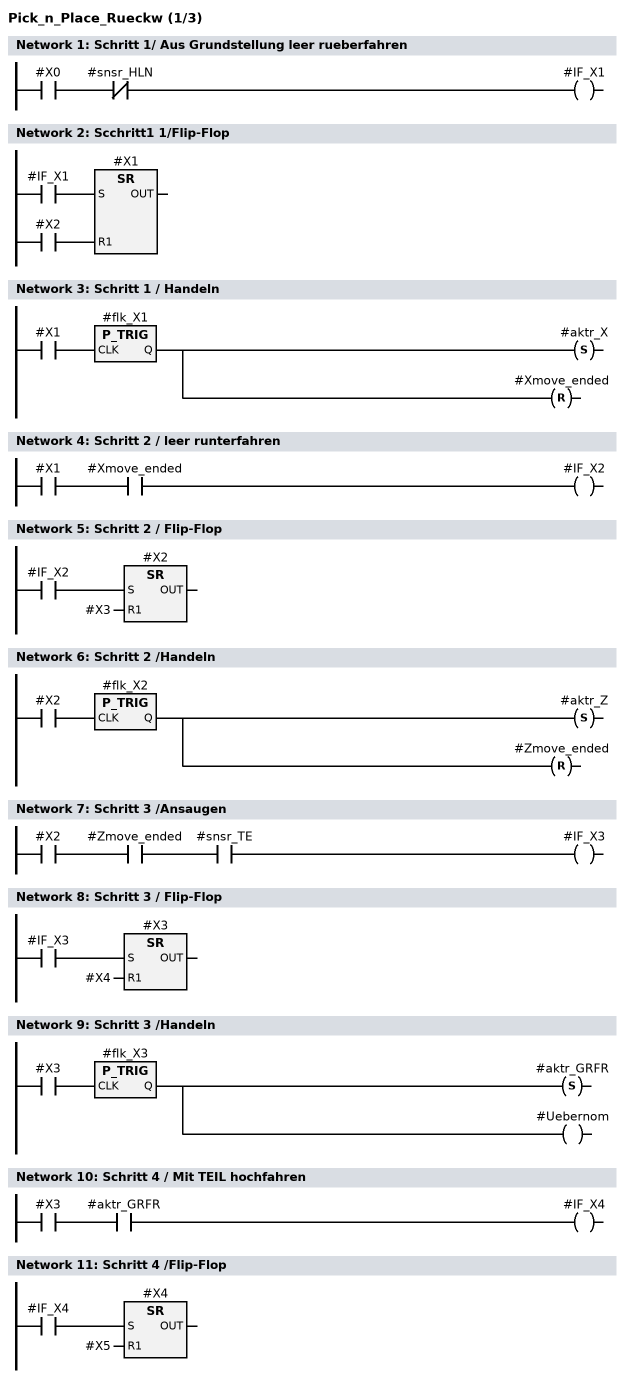
   RUNG wire#powerrail
      Contact( #X0 )
      I_Contact( #snsr_HLN )
      Coil( #IF_X1 )
   END_RUNG
   // the same network as SCL:
   #IF_X1 := #X0 AND NOT #snsr_HLN;
END_REGION

REGION Network 2: Scchritt1 1/Flip-Flop
   RUNG wire#powerrail
      Contact( #IF_X1 )
      S_SR(operand := #X1, r1 := wire#w1)
   END_RUNG
   RUNG wire#powerrail
      Contact( #X2 )
   END_RUNG wire#w1
   // the same network as SCL:
   IF #IF_X1 THEN
       #X1 := TRUE;   // SR flip-flop
   END_IF;
   IF #X2 THEN #X1 := FALSE; END_IF;
END_REGION

REGION Network 3: Schritt 1 / Handeln
   RUNG wire#powerrail
      Contact( #X1 )
      P_Trig( #flk_X1 )
      wire#w1
      S_Coil( #aktr_X )
   END_RUNG
   RUNG wire#w1
      R_Coil( #Xmove_ended )
   END_RUNG
   // the same network as SCL:
   #_w1 := #X1 AND NOT #flk_X1;   // rising edge
   #flk_X1 := #X1;
   IF #_w1 THEN
       #aktr_X := TRUE;
       #Xmove_ended := FALSE;
   END_IF;
END_REGION

REGION Network 4: Schritt 2 / leer runterfahren
   RUNG wire#powerrail
      Contact( #X1 )
      Contact( #Xmove_ended )
      Coil( #IF_X2 )
   END_RUNG
   // the same network as SCL:
   #IF_X2 := #X1 AND #Xmove_ended;
END_REGION

REGION Network 5: Schritt 2 / Flip-Flop
   RUNG wire#powerrail
      Contact( #IF_X2 )
      S_SR(operand := #X2, r1 := #X3)
   END_RUNG
   // the same network as SCL:
   IF #IF_X2 THEN
       #X2 := TRUE;   // SR flip-flop
   END_IF;
   IF #X3 THEN #X2 := FALSE; END_IF;
END_REGION

REGION Network 6: Schritt 2 /Handeln
   RUNG wire#powerrail
      Contact( #X2 )
      P_Trig( #flk_X2 )
      wire#w1
      S_Coil( #aktr_Z )
   END_RUNG
   RUNG wire#w1
      R_Coil( #Zmove_ended )
   END_RUNG
   // the same network as SCL:
   #_w1 := #X2 AND NOT #flk_X2;   // rising edge
   #flk_X2 := #X2;
   IF #_w1 THEN
       #aktr_Z := TRUE;
       #Zmove_ended := FALSE;
   END_IF;
END_REGION

REGION Network 7: Schritt 3 /Ansaugen
   RUNG wire#powerrail
      Contact( #X2 )
      Contact( #Zmove_ended )
      Contact( #snsr_TE )
      Coil( #IF_X3 )
   END_RUNG
   // the same network as SCL:
   #IF_X3 := #X2 AND #Zmove_ended AND #snsr_TE;
END_REGION

REGION Network 8: Schritt 3 / Flip-Flop
   RUNG wire#powerrail
      Contact( #IF_X3 )
      S_SR(operand := #X3, r1 := #X4)
   END_RUNG
   // the same network as SCL:
   IF #IF_X3 THEN
       #X3 := TRUE;   // SR flip-flop
   END_IF;
   IF #X4 THEN #X3 := FALSE; END_IF;
END_REGION

REGION Network 9: Schritt 3 /Handeln
   RUNG wire#powerrail
      Contact( #X3 )
      P_Trig( #flk_X3 )
      wire#w1
      S_Coil( #aktr_GRFR )
   END_RUNG
   RUNG wire#w1
      Coil( #Uebernom )
   END_RUNG
   // the same network as SCL:
   #_w1 := #X3 AND NOT #flk_X3;   // rising edge
   #flk_X3 := #X3;
   IF #_w1 THEN #aktr_GRFR := TRUE; END_IF;
   #Uebernom := #_w1;
END_REGION

REGION Network 10: Schritt 4 / Mit TEIL hochfahren
   RUNG wire#powerrail
      Contact( #X3 )
      Contact( #aktr_GRFR )
      Coil( #IF_X4 )
   END_RUNG
   // the same network as SCL:
   #IF_X4 := #X3 AND #aktr_GRFR;
END_REGION

REGION Network 11: Schritt 4 /Flip-Flop
   RUNG wire#powerrail
      Contact( #IF_X4 )
      S_SR(operand := #X4, r1 := #X5)
   END_RUNG
   // the same network as SCL:
   IF #IF_X4 THEN
       #X4 := TRUE;   // SR flip-flop
   END_IF;
   IF #X5 THEN #X4 := FALSE; END_IF;
END_REGION

REGION Network 12: Schritt 4 / Handeln
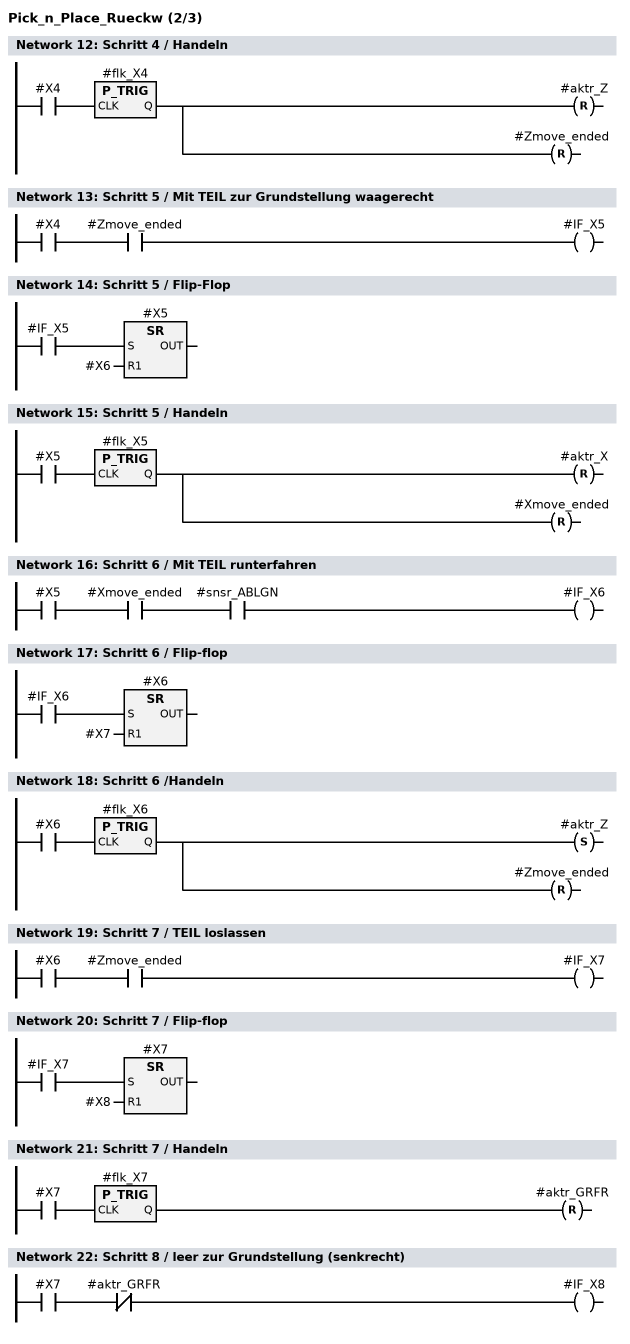
   RUNG wire#powerrail
      Contact( #X4 )
      P_Trig( #flk_X4 )
      wire#w1
      R_Coil( #aktr_Z )
   END_RUNG
   RUNG wire#w1
      R_Coil( #Zmove_ended )
   END_RUNG
   // the same network as SCL:
   #_w1 := #X4 AND NOT #flk_X4;   // rising edge
   #flk_X4 := #X4;
   IF #_w1 THEN
       #aktr_Z := FALSE;
       #Zmove_ended := FALSE;
   END_IF;
END_REGION

REGION Network 13: Schritt 5 / Mit TEIL zur Grundstellung waagerecht
   RUNG wire#powerrail
      Contact( #X4 )
      Contact( #Zmove_ended )
      Coil( #IF_X5 )
   END_RUNG
   // the same network as SCL:
   #IF_X5 := #X4 AND #Zmove_ended;
END_REGION

REGION Network 14: Schritt 5 / Flip-Flop
   RUNG wire#powerrail
      Contact( #IF_X5 )
      S_SR(operand := #X5, r1 := #X6)
   END_RUNG
   // the same network as SCL:
   IF #IF_X5 THEN
       #X5 := TRUE;   // SR flip-flop
   END_IF;
   IF #X6 THEN #X5 := FALSE; END_IF;
END_REGION

REGION Network 15: Schritt 5 / Handeln
   RUNG wire#powerrail
      Contact( #X5 )
      P_Trig( #flk_X5 )
      wire#w1
      R_Coil( #aktr_X )
   END_RUNG
   RUNG wire#w1
      R_Coil( #Xmove_ended )
   END_RUNG
   // the same network as SCL:
   #_w1 := #X5 AND NOT #flk_X5;   // rising edge
   #flk_X5 := #X5;
   IF #_w1 THEN
       #aktr_X := FALSE;
       #Xmove_ended := FALSE;
   END_IF;
END_REGION

REGION Network 16: Schritt 6 / Mit TEIL runterfahren
   RUNG wire#powerrail
      Contact( #X5 )
      Contact( #Xmove_ended )
      Contact( #snsr_ABLGN )
      Coil( #IF_X6 )
   END_RUNG
   // the same network as SCL:
   #IF_X6 := #X5 AND #Xmove_ended AND #snsr_ABLGN;
END_REGION

REGION Network 17: Schritt 6 / Flip-flop
   RUNG wire#powerrail
      Contact( #IF_X6 )
      S_SR(operand := #X6, r1 := #X7)
   END_RUNG
   // the same network as SCL:
   IF #IF_X6 THEN
       #X6 := TRUE;   // SR flip-flop
   END_IF;
   IF #X7 THEN #X6 := FALSE; END_IF;
END_REGION

REGION Network 18: Schritt 6 /Handeln
   RUNG wire#powerrail
      Contact( #X6 )
      P_Trig( #flk_X6 )
      wire#w1
      S_Coil( #aktr_Z )
   END_RUNG
   RUNG wire#w1
      R_Coil( #Zmove_ended )
   END_RUNG
   // the same network as SCL:
   #_w1 := #X6 AND NOT #flk_X6;   // rising edge
   #flk_X6 := #X6;
   IF #_w1 THEN
       #aktr_Z := TRUE;
       #Zmove_ended := FALSE;
   END_IF;
END_REGION

REGION Network 19: Schritt 7 / TEIL loslassen
   RUNG wire#powerrail
      Contact( #X6 )
      Contact( #Zmove_ended )
      Coil( #IF_X7 )
   END_RUNG
   // the same network as SCL:
   #IF_X7 := #X6 AND #Zmove_ended;
END_REGION

REGION Network 20: Schritt 7 / Flip-flop
   RUNG wire#powerrail
      Contact( #IF_X7 )
      S_SR(operand := #X7, r1 := #X8)
   END_RUNG
   // the same network as SCL:
   IF #IF_X7 THEN
       #X7 := TRUE;   // SR flip-flop
   END_IF;
   IF #X8 THEN #X7 := FALSE; END_IF;
END_REGION

REGION Network 21: Schritt 7 / Handeln
   RUNG wire#powerrail
      Contact( #X7 )
      P_Trig( #flk_X7 )
      R_Coil( #aktr_GRFR )
   END_RUNG
   // the same network as SCL:
   #_w1 := #X7 AND NOT #flk_X7;   // rising edge
   #flk_X7 := #X7;
   IF #_w1 THEN #aktr_GRFR := FALSE; END_IF;
END_REGION

REGION Network 22: Schritt 8 / leer zur Grundstellung (senkrecht)
   RUNG wire#powerrail
      Contact( #X7 )
      I_Contact( #aktr_GRFR )
      Coil( #IF_X8 )
   END_RUNG
   // the same network as SCL:
   #IF_X8 := #X7 AND NOT #aktr_GRFR;
END_REGION

REGION Network 23: Schritt 8 / Flip-Flop
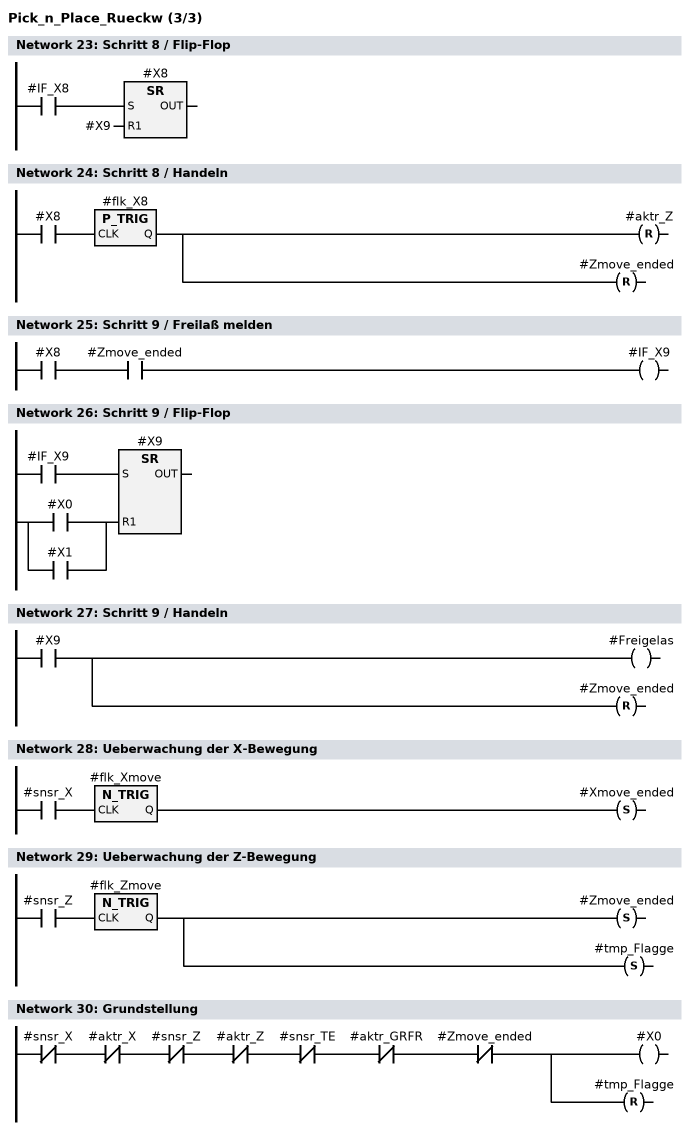
   RUNG wire#powerrail
      Contact( #IF_X8 )
      S_SR(operand := #X8, r1 := #X9)
   END_RUNG
   // the same network as SCL:
   IF #IF_X8 THEN
       #X8 := TRUE;   // SR flip-flop
   END_IF;
   IF #X9 THEN #X8 := FALSE; END_IF;
END_REGION

REGION Network 24: Schritt 8 / Handeln
   RUNG wire#powerrail
      Contact( #X8 )
      P_Trig( #flk_X8 )
      wire#w1
      R_Coil( #aktr_Z )
   END_RUNG
   RUNG wire#w1
      R_Coil( #Zmove_ended )
   END_RUNG
   // the same network as SCL:
   #_w1 := #X8 AND NOT #flk_X8;   // rising edge
   #flk_X8 := #X8;
   IF #_w1 THEN
       #aktr_Z := FALSE;
       #Zmove_ended := FALSE;
   END_IF;
END_REGION

REGION Network 25: Schritt 9 / Freilaß melden
   RUNG wire#powerrail
      Contact( #X8 )
      Contact( #Zmove_ended )
      Coil( #IF_X9 )
   END_RUNG
   // the same network as SCL:
   #IF_X9 := #X8 AND #Zmove_ended;
END_REGION

REGION Network 26: Schritt 9 / Flip-Flop
   RUNG wire#powerrail
      Contact( #IF_X9 )
      S_SR(operand := #X9, r1 := wire#w1)
   END_RUNG
   RUNG wire#powerrail
      Contact( #X0 )
   END_RUNG wire#w1
   RUNG wire#powerrail
      Contact( #X1 )
   END_RUNG wire#w1
   // the same network as SCL:
   IF #IF_X9 THEN
       #X9 := TRUE;   // SR flip-flop
   END_IF;
   IF #X0 OR #X1 THEN #X9 := FALSE; END_IF;
END_REGION

REGION Network 27: Schritt 9 / Handeln
   RUNG wire#powerrail
      Contact( #X9 )
      wire#w1
      Coil( #Freigelas )
   END_RUNG
   RUNG wire#w1
      R_Coil( #Zmove_ended )
   END_RUNG
   // the same network as SCL:
   #Freigelas := #X9;
   IF #X9 THEN #Zmove_ended := FALSE; END_IF;
END_REGION

REGION Network 28: Ueberwachung der X-Bewegung
   RUNG wire#powerrail
      Contact( #snsr_X )
      N_Trig( #flk_Xmove )
      S_Coil( #Xmove_ended )
   END_RUNG
   // the same network as SCL:
   #_w1 := NOT #snsr_X AND #flk_Xmove;   // falling edge
   #flk_Xmove := #snsr_X;
   IF #_w1 THEN #Xmove_ended := TRUE; END_IF;
END_REGION

REGION Network 29: Ueberwachung der Z-Bewegung
   RUNG wire#powerrail
      Contact( #snsr_Z )
      N_Trig( #flk_Zmove )
      wire#w1
      S_Coil( #Zmove_ended )
   END_RUNG
   RUNG wire#w1
      S_Coil( #tmp_Flagge )
   END_RUNG
   // the same network as SCL:
   #_w1 := NOT #snsr_Z AND #flk_Zmove;   // falling edge
   #flk_Zmove := #snsr_Z;
   IF #_w1 THEN
       #Zmove_ended := TRUE;
       #tmp_Flagge := TRUE;
   END_IF;
END_REGION

REGION Network 30: Grundstellung
   RUNG wire#powerrail
      I_Contact( #snsr_X )
      I_Contact( #aktr_X )
      I_Contact( #snsr_Z )
      I_Contact( #aktr_Z )
      I_Contact( #snsr_TE )
      I_Contact( #aktr_GRFR )
      I_Contact( #Zmove_ended )
      wire#w1
      Coil( #X0 )
   END_RUNG
   RUNG wire#w1
      R_Coil( #tmp_Flagge )
   END_RUNG
   // the same network as SCL:
   #X0 := NOT #snsr_X AND NOT #aktr_X AND NOT #snsr_Z AND NOT #aktr_Z AND NOT #snsr_TE AND NOT #aktr_GRFR AND NOT #Zmove_ended;
   IF #X0 THEN #tmp_Flagge := FALSE; END_IF;
END_REGION
END_FUNCTION_BLOCK

FUNCTION "04_Kommisionierung" : Void   // FC1, FBD
TITLE = Automatikbetrieb für das Project 04-Kommisionierung mit Factory IO
{ S7_Optimized_Access := 'FALSE' }
VERSION : 0.1
// Das Programm gewährleistet NUR AUTOMATK-Betrieb OHNE Beachtung NOT-HALT und Schalter EIN/AUS. Muss separat realisiert werden (ist vom mir in "03-Fertigung" entwickelt). Für den Pick-and-Place Manipulator muss zusätzlicht zu den Schritten eine Bedinung hinzugefügt werden, die prüft, ob NOT-HALT aktiv ist, falls dann darf der nächster Schrit nicht aktiviert werden, eigentlich ganz einfache Änderung.
BEGIN

REGION Network 1: 04-00 Kistenerzeugung
   // Hier werden die Kisten dauernd erzeugt sobald das erste Band frei ist und abwechslend markiert für die nähre und ferne Ladestation
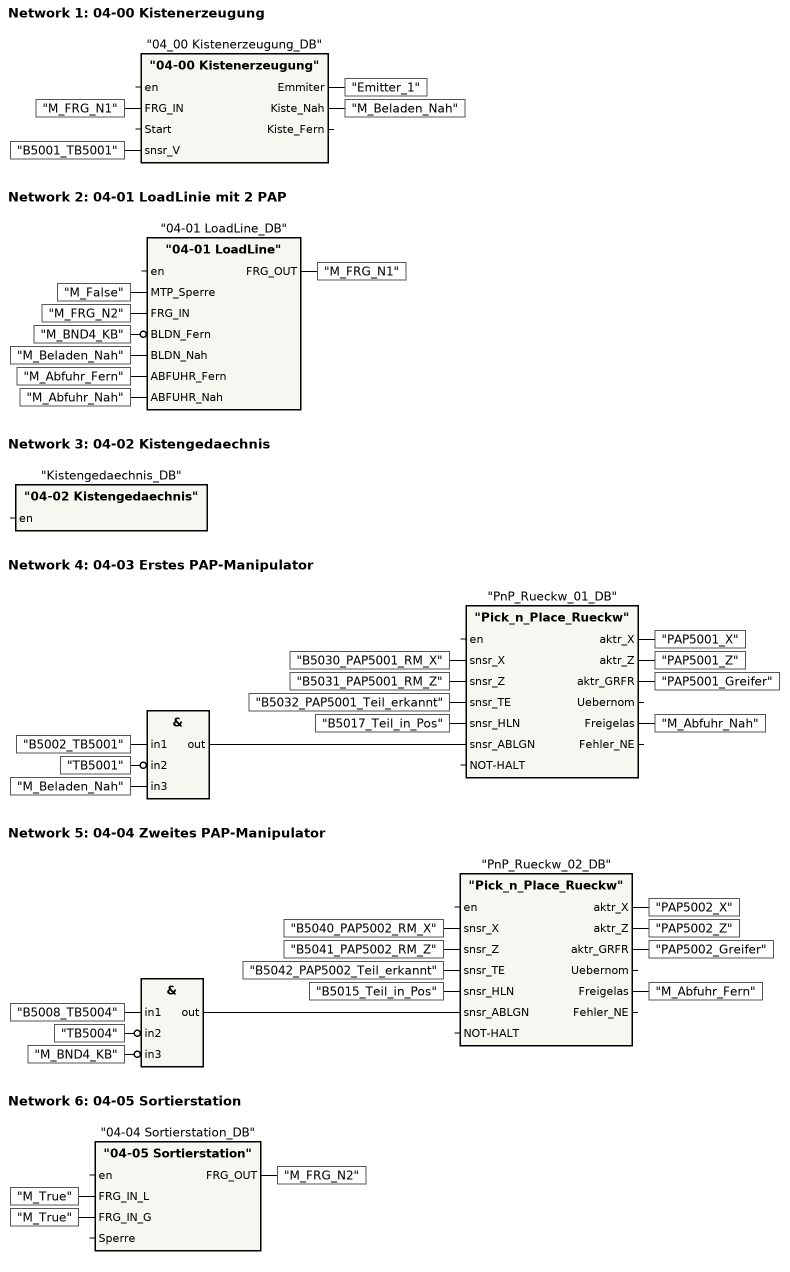
   "04_00 Kistenerzeugung_DB"(FRG_IN := "M_FRG_N1",   // "04-00 Kistenerzeugung"
                           snsr_V := "B5001_TB5001",
                           Emmiter => "Emitter_1",
                           Kiste_Nah => "M_Beladen_Nah");
END_REGION

REGION Network 2: 04-01 LoadLinie mit 2 PAP
   // Die Reihe von Förderbenden, wo die leere Kisten mit den Teilen beladen werden und zur Sortierstation weitergegeben
   "04-01 LoadLine_DB"(MTP_Sperre := "M_False",   // "04-01 LoadLine"
                       FRG_IN := "M_FRG_N2",
                       BLDN_Fern := NOT "M_BND4_KB",
                       BLDN_Nah := "M_Beladen_Nah",
                       ABFUHR_Fern := "M_Abfuhr_Fern",
                       ABFUHR_Nah := "M_Abfuhr_Nah",
                       FRG_OUT => "M_FRG_N1");
END_REGION

REGION Network 3: 04-02 Kistengedaechnis
   // Hier wird der Status (beladen/leer) jeder Kiste gespeichert zwischen beined Ladestationen
   "Kistengedaechnis_DB"();   // "04-02 Kistengedaechnis"
END_REGION

REGION Network 4: 04-03 Erstes PAP-Manipulator
   // Schrittkettenprogramm für den ersten PAP
   "PnP_Rueckw_01_DB"(snsr_X := "B5030_PAP5001_RM_X",   // "Pick_n_Place_Rueckw"
                      snsr_Z := "B5031_PAP5001_RM_Z",
                      snsr_TE := "B5032_PAP5001_Teil_erkannt",
                      snsr_HLN := "B5017_Teil_in_Pos",
                      snsr_ABLGN := "B5002_TB5001" AND NOT "TB5001" AND "M_Beladen_Nah",
                      aktr_X => "PAP5001_X",
                      aktr_Z => "PAP5001_Z",
                      aktr_GRFR => "PAP5001_Greifer",
                      Freigelas => "M_Abfuhr_Nah");
END_REGION

REGION Network 5: 04-04 Zweites PAP-Manipulator
   // Schrittkettenprogramm für den zweiten PAP
   "PnP_Rueckw_02_DB"(snsr_X := "B5040_PAP5002_RM_X",   // "Pick_n_Place_Rueckw"
                      snsr_Z := "B5041_PAP5002_RM_Z",
                      snsr_TE := "B5042_PAP5002_Teil_erkannt",
                      snsr_HLN := "B5015_Teil_in_Pos",
                      snsr_ABLGN := "B5008_TB5004" AND NOT "TB5004" AND NOT "M_BND4_KB",
                      aktr_X => "PAP5002_X",
                      aktr_Z => "PAP5002_Z",
                      aktr_GRFR => "PAP5002_Greifer",
                      Freigelas => "M_Abfuhr_Fern");
END_REGION

REGION Network 6: 04-05 Sortierstation
   "04-04 Sortierstation_DB"(FRG_IN_L := "M_True", FRG_IN_G := "M_True", FRG_OUT => "M_FRG_N2");   // "04-05 Sortierstation"
END_REGION
END_FUNCTION

ORGANIZATION_BLOCK "Main"   // OB1, FBD
TITLE = "Main Program Sweep (Cycle)"
{ S7_Optimized_Access := 'FALSE' }
VERSION : 0.1
   VAR_TEMP
      OB1_EV_CLASS : Byte;   // Bits 0-3 = 1 (Coming event), Bits 4-7 = 1 (Event class 1)
      OB1_SCAN_1 : Byte;   // 1 (Cold restart scan 1 of OB 1), 3 (Scan 2-n of OB 1)
      OB1_PRIORITY : Byte;   // Priority of OB Execution
      OB1_OB_NUMBR : Byte;   // 1 (Organization block 1, OB1)
      OB1_RESERVED_1 : Byte;   // Reserved for system
      OB1_RESERVED_2 : Byte;   // Reserved for system
      OB1_PREV_CYCLE : Int;   // Cycle time of previous OB1 scan (milliseconds)
      OB1_MIN_CYCLE : Int;   // Minimum cycle time of OB1 (milliseconds)
      OB1_MAX_CYCLE : Int;   // Maximum cycle time of OB1 (milliseconds)
      OB1_DATE_TIME : Date_And_Time;   // Date and time OB1 started
   END_VAR
BEGIN

REGION Network 1: Merker Immer_TRUE initialisieren
   // Werden für provisoriesche Zwecke benutzt, bei der Integration im gesammten Programm müssen ersetzt werden!!!
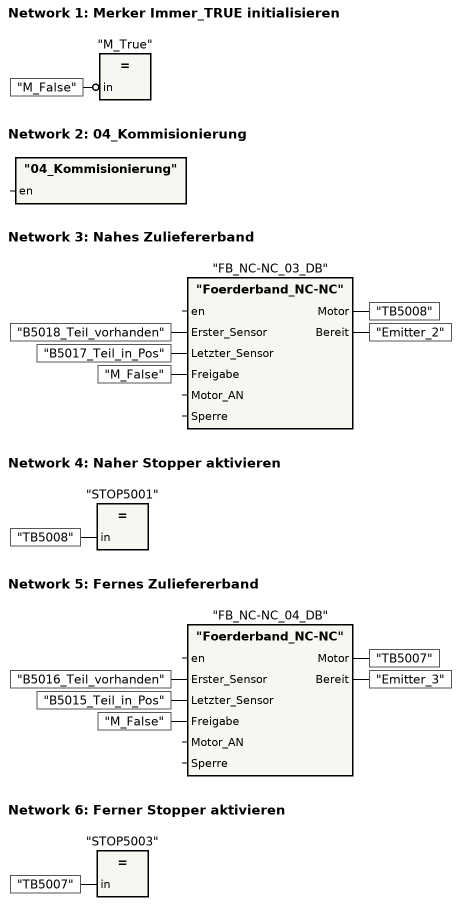
   "M_True" := NOT "M_False";
END_REGION

REGION Network 2: 04_Kommisionierung
   // Aufruf AUTOmatik-Betrieb der Kommisionierungslinie OHNE Behandlung von Fehler
   "04_Kommisionierung"();
END_REGION

REGION Network 3: Nahes Zuliefererband
   // führt blaue Teile zur erster Ladestation, bei der Integration im gesammten Programm müssen ersetzt werden!!!
   "FB_NC-NC_03_DB"(Erster_Sensor := "B5018_Teil_vorhanden",   // "Foerderband_NC-NC"
                    Letzter_Sensor := "B5017_Teil_in_Pos",
                    Freigabe := "M_False",
                    Motor => "TB5008",
                    Bereit => "Emitter_2");
END_REGION

REGION Network 4: Naher Stopper aktivieren
   // bei der Integration im gesammten Programm müssen ersetzt werden!!!
   "STOP5001" := "TB5008";
END_REGION

REGION Network 5: Fernes Zuliefererband
   // führt blaue Teile zur erster Ladestation, bei der Integration im gesammten Programm müssen ersetzt werden!!!
   "FB_NC-NC_04_DB"(Erster_Sensor := "B5016_Teil_vorhanden",   // "Foerderband_NC-NC"
                    Letzter_Sensor := "B5015_Teil_in_Pos",
                    Freigabe := "M_False",
                    Motor => "TB5007",
                    Bereit => "Emitter_3");
END_REGION

REGION Network 6: Ferner Stopper aktivieren
   // bei der Integration im gesammten Programm müssen ersetzt werden!!!
   "STOP5003" := "TB5007";
END_REGION
END_ORGANIZATION_BLOCK

// ===== library: MasterCopy "RB_TB_einfach" =====

FUNCTION_BLOCK "RB_TB_einfach"   // FB101, GRAPH
{ S7_Optimized_Access := 'FALSE' }
VERSION : 0.1
// Einfacher Steuerbaustein RB / TB 
// Sensor Anfang / Ende  NO
   VAR_INPUT
      INIT_SQ : Bool := false;   // Kette in Initialzustand versetzen
      A_EIN : Bool;
      A_NOT_HALT : Bool;
      Nachfolgendes_Agg_frei : Bool;
      Sensor_vorheriges_Agg : Bool;
      Sensor_Anfang : Bool;   // Öffner
      Sensor_Ende : Bool;   // Öffner
   END_VAR
   VAR_OUTPUT
      Schritt_Nummer : Int;
      Aggregat : Bool;
      Aggregat_frei : Bool;
   END_VAR
   VAR
      HM_FLAM : Array[1..8] of Bool;
      Flanke : Array[1..8] of Bool;
      HM_Agg_Frei : Bool;
      HM_belegt : Bool;
      SWITCH : Array[0..0] of DWord;
      SW_SQTS : Array[0..6] of Byte;
      SW_ADDR : Word := 16#C;
      G7T_0 : GraphTransition;
      G7S_0 : GraphStep;
      PRE_CRIT : Array[0..1] of DWord;
      POST_CRIT : Array[0..0] of DWord;
      TVX : Array[0..2] of Byte;
      TTX : Array[0..2] of Byte;
      TSX : Array[0..2] of Byte;
      S00X : Array[0..2] of Byte;
      SOFFX : Array[0..2] of Byte;
      SONX : Array[0..2] of Byte;
      SAX : Array[0..2] of Byte;
      SERRX : Array[0..7] of Byte;
      SMX : Array[0..7] of Byte;
      S0X : Array[0..7] of Byte;
      S1X : Array[0..7] of Byte;
      S_DISPLAY : Int;   // Interne Anzeige des Ausgangsparameters S_NO
      S_SEL_OLD : Int;   // Vorheriger Wert an S_SEL
      S_DISPIDX : Byte;   // Index des Schritts, der an S_NO anliegt
      T_DISPIDX : Byte;   // Index der Transition, die an T_NO anliegt
      MOPEDGE : Struct
         AUTO : Bool := false;
         MAN : Bool := false;
         TAP : Bool := false;
         TOP : Bool := false;
         ACK_S : Bool := false;
         REG_S : Bool := false;
         T_PREV : Bool := false;
         T_NEXT : Bool := false;
         LOCK : Bool := false;
         SUP : Bool := false;
         ACKREQ : Bool := false;
         SSKIP : Bool := false;
         OFF : Bool := false;
         INIT : Bool := false;
         HALT : Bool := false;
         TMS_HALT : Bool := false;
         OPS_ZERO : Bool := false;
         SACT_DISP : Bool := false;
         SEF_DISP : Bool := false;
         SALL_DISP : Bool := false;
         S_PREV : Bool := false;
         S_NEXT : Bool := false;
         S_SELOK : Bool := false;
         S_ON : Bool := false;
         S_OFF : Bool := false;
         T_PUSH : Bool := false;
         REG : Bool := false;
         ACK : Bool := false;
         IL_PERM : Bool := false;
         T_PERM : Bool := false;
         ILP_MAN : Bool := false;
      END_STRUCT;
      MOP : Struct   // Betriebsart
         AUTO : Bool := true;   // Zustand: Automatischer Betrieb
         MAN : Bool := false;   // Zustand: Handbetrieb
         TAP : Bool := false;   // Zustand: Halbautomatisch/Weiterschalten mit Transition
         TOP : Bool := false;   // Zustand: Halbautomatisch/Ignoriere Transition
         ACK_S : Bool := false;   // Anforderung: Schritt quittieren, der an Parameter S_NO anliegt
         REG_S : Bool := false;   // Anforderung: Schritt registrieren, der an Parameter S_NO anliegt
         T_PREV : Bool := false;   // Anforderung: Vorherige gültige Transition am Parameter T_NO ausgeben
         T_NEXT : Bool := false;   // Anforderung: Nächste gültige Transition am Parameter T_NO ausgeben
         LOCK : Bool := true;   // Zustand: Interlockbearbeitung aktiviert
         SUP : Bool := true;   // Zustand: Supervisionsbearbeitung aktiviert
         ACKREQ : Bool := false;   // Zustand: Quittierung erforderlich
         SSKIP : Bool := false;   // Zustand: "Schritte überspringen" aktiviert
         OFF : Bool := false;   // Anforderung: Alle Schritte deaktivieren
         INIT : Bool := true;   // Anforderung: Kette in Initialzustand schalten
         HALT : Bool := false;   // Zustand: Kette schaltet nicht weiter
         TMS_HALT : Bool := false;   // Zustand: Alle internen Zeiten angehalten
         OPS_ZERO : Bool := false;   // Zustand: Alle mit N, L, D bearbeitete Operanden auf 0 gesetzt
         SACT_DISP : Bool := true;   // Zustand: Nur aktive Schritte anzeigen
         SEF_DISP : Bool := false;   // Zustand: Nur fehlerhafte und gestörte Schritte anzeigen
         SALL_DISP : Bool := false;   // Zustand: Alle Schritte anzeigen
         S_PREV : Bool := false;   // Anforderung: Vorherigen Schritt am Parameter S_NO ausgeben
         S_NEXT : Bool := false;   // Anforderung: Nächsten Schritt am Parameter S_NO ausgeben
         S_SELOK : Bool := false;   // Anforderung: Schrittnummer, die am Parameter S_SEL anliegt, am Parameter S_NO ausgeben
         S_ON : Bool := false;   // Anforderung: Schritt aktivieren, der am Parameter S_NO anliegt
         S_OFF : Bool := false;   // Anforderung: Schritt deaktivieren, der am Parameter S_NO anliegt
         T_PUSH : Bool := false;   // Anforderung: Schaltfreigabe für Transition
         REG : Bool := false;   // Anforderung: Alle Interlock- und Supervisionsfehler registrieren
         ACK : Bool := false;   // Anforderung: Alle Interlock- und Supervisionsfehler quittieren
         IL_PERM : Bool := false;   // Zustand: Permanente Bearbeitung aller Interlocks
         T_PERM : Bool := false;   // Zustand: Permanente Bearbeitung aller Transitionen
         ILP_MAN : Bool := false;   // Zustand: Permanente Bearbeitung aller Interlocks im Handbetrieb
      END_STRUCT;
      TICKS : Struct   // Zeittakte
         DELTA : Time := T#0ms;   // Zeitdifferenz zwischen zwei Zyklen
         OLD : Time := T#0ms;   // 10 ms Taktzählerstand im letzten Zyklus
         NEW : Time := T#0ms;   // 10 ms Taktzählerstand in diesem Zyklus
      END_STRUCT;
      SQ_FLAGS : Struct   // Kettenmerker
         ERR_FLT : Bool := false;   // Sammelfehler Interlock und Supervision
         ERROR : Bool := false;   // Sammelfehler Interlock
         FAULT : Bool := false;   // Sammelfehler Supervision
         RT_FAIL : Bool := false;   // Laufzeitfehler
         NO_SNO : Bool := false;   // Angeforderte Schrittnummer nicht gefunden
         NF_OFL : Bool := false;   // Überlauf: Zu viele Anforderungen ON oder OFF
         SA_OFL : Bool := false;   // Überlauf: Zu viele Schritte aktiv
         TV_OFL : Bool := false;   // Überlauf: Zu viele gültige Transitionen
         MSG_OFL : Bool := false;   // Überlauf: Nicht genügend Systemressourcen fü ALARM_S
         NO_SWI : Bool := false;   // Nicht Schalten in diesem Zyklus
         CYC_OP : Bool := false;   // Zyklische Bearbeitung der Kette nach Initialisierung
         AS_MSG : Bool := true;   // Meldungen zur Laufzeit durch Anweisung aktiviert oder deaktiviert
         AS_SEND : Bool := false;   // Meldungen von WR_USMSG senden oder nur in Diagnosepuffer eintragen
         SQ_BUSY : Bool := false;   // Interner Flankenmerker für Vorgangsbearbeitung
         SA_BUSY : Bool := false;   // Interner Flankenmerker für Vorgangsbearbeitung
         AS_SIG : Bool := false;   // Flankenmerker für Meldungen von Alarm_S und Alarm_SQ
      END_STRUCT;
      S_PTR : DWord := 16#450;
      S_PTR2 : DWord := 16#0;
      S_PTR3 : DWord := 16#D50;
      S_PTR4 : DWord := 16#D10;
      T_PTR : DWord := 16#CD0;
      C_AR2 : DWord := 16#0;
      M_FBDB : DWord := 16#640000;
      M_SNO : Word := 16#4;
      M_EVID : Word := 16#0;
      M_EVIL : C_Alarm_s;
      M_EVSV : C_Alarm_s;
      M_EV : DWord := 16#C30;
      CRIT : Array[0..31] of Bool;
      S_START : Byte := 16#0;
      S_IDX : Byte := 16#0;
      S_INT : Int := 72;
      S_TMP : Byte := 16#0;
      T_START : Byte := 16#0;
      T_IDX : Byte := 16#0;
      T_TMP : Byte := 16#0;
      T_TMP2 : Byte := 16#00;
      TV_POT : Byte := 16#02;
      RETURN1 : Byte := 16#0;
      RETURN2 : Byte := 16#0;
      SINI : Array[0..2] of Byte;
      LSTT : Array[0..6] of Byte;
      ATAJ : Array[0..6] of Byte;
      ATAB : Array[0..6] of Byte;
      PSTT : Array[0..6] of Byte;
      NSTT : Array[0..6] of Byte;
      ASSJ : Array[0..6] of Byte;
      ASSB : Array[0..6] of Byte;
      PTTS : Array[0..6] of Byte;
      NTTS : Array[0..6] of Byte;
      PRE_CNT : Word := 16#2;
      POST_CNT : Word := 16#1;
      ADR_COND : Word := 16#0;
      MAX_TVAL : Byte := 16#1;
      MAX_SACT : Byte := 16#1;
      MAX_CRIT : Byte := 16#4;
      T_CNT : Byte := 16#6;
      SUP_CNT : Byte := 16#0;
      LOCK_CNT : Byte := 16#5;
      S_CNT : Byte := 16#6;
      SQ_CNT : Byte := 16#1;
      PRS_INPAR : DWord := 16#40000000;
      PRS_OUTPAR : DWord := 16#0;
      GC_FLAGS : Struct
         T_MACH : Byte := 16#EB;
         COND_ED : Byte := 16#E2;
         W_LEVEL : Byte := 16#D5;
         FB_IF : Byte := 16#FA;
         AS_MSG : Word := 16#404;
         SSB : Word := 16#108;
         DILG : Word := 16#27E;
         ADDR_T0 : Word := 16#1A;
         CRIT_AVAIL : Bool := false;
         SSKIP_AVAIL : Bool := true;
         SSKIP_ON : Bool := false;
         ACK_REQ : Bool := false;
         SYNC_AVAIL : Bool := true;
         ILP_MAN : Bool := false;
         SWM_LOCKED : Bool := false;
         SAVE_SW : Bool := true;
      END_STRUCT;
      G7_FBMARK : Byte := 16#3C;
      G7_RELEASE : Byte := 16#3C;
      G7_ID2 : Byte := 16#37;
      G7_ID1 : Byte := 16#47;
   END_VAR
   // SW_SQTS[0] := 16#1;
   // TVX[0] := 16#1;
   // TTX[0] := 16#1;
   // TSX[0] := 16#1;
   // S00X[0] := 16#1;
   // SOFFX[0] := 16#1;
   // SONX[0] := 16#1;
   // SAX[0] := 16#1;
   // SERRX[0] := 16#1;
   // SMX[0] := 16#1;
   // S0X[0] := 16#1;
   // S1X[0] := 16#1;
   // SINI[0] := 16#2;
   // SINI[1] := 16#1;
   // SINI[2] := 0;
   // LSTT[0] := 0;
   // LSTT[1] := 0;
   // LSTT[2] := 0;
   // LSTT[3] := 0;
   // LSTT[4] := 0;
   // LSTT[5] := 0;
   // ATAJ[0] := 0;
   // ATAJ[1] := 16#1;
   // ATAJ[2] := 16#2;
   // ATAJ[3] := 16#3;
   // ATAJ[4] := 16#4;
   // ATAJ[5] := 16#5;
   // ATAB[0] := 0;
   // ATAB[1] := 16#1;
   // ATAB[2] := 16#2;
   // ATAB[3] := 16#3;
   // ATAB[4] := 16#4;
   // ATAB[5] := 16#5;
   // PSTT[0] := 0;
   // PSTT[1] := 16#1;
   // PSTT[2] := 16#2;
   // PSTT[3] := 16#3;
   // PSTT[4] := 16#4;
   // PSTT[5] := 16#5;
   // NSTT[0] := 16#1;
   // NSTT[1] := 16#2;
   // NSTT[2] := 16#3;
   // NSTT[3] := 16#4;
   // NSTT[4] := 16#5;
   // NSTT[5] := 16#6;
   // ASSJ[0] := 0;
   // ASSJ[1] := 16#1;
   // ASSJ[2] := 16#2;
   // ASSJ[3] := 16#3;
   // ASSJ[4] := 16#4;
   // ASSJ[5] := 16#5;
   // ASSB[0] := 0;
   // ASSB[1] := 16#1;
   // ASSB[2] := 16#2;
   // ASSB[3] := 16#3;
   // ASSB[4] := 16#4;
   // ASSB[5] := 16#5;
   // PTTS[0] := 0;
   // PTTS[2] := 16#1;
   // PTTS[3] := 16#2;
   // PTTS[4] := 16#3;
   // PTTS[5] := 16#4;
   // NTTS[0] := 0;
   // NTTS[1] := 16#1;
   // NTTS[2] := 16#2;
   // NTTS[3] := 16#3;
   // NTTS[4] := 16#4;
   // NTTS[5] := 16#5;
   // LSTT[6] := 16#1;
   // ATAJ[6] := 16#6;
   // ATAB[6] := 16#6;
   // PSTT[6] := 16#6;
   // NSTT[6] := 16#1;
   // ASSJ[6] := 16#6;
   // ASSB[6] := 16#6;
   // PTTS[6] := 16#5;
   // NTTS[6] := 16#6;
BEGIN
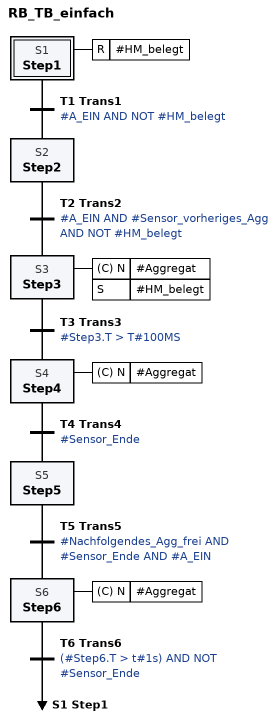
   // permanent pre-instructions
   NETWORK 1
      #HM_Agg_Frei := NOT #HM_belegt;
      #Aggregat_frei := NOT #HM_belegt;
   NETWORK 2
   TITLE = Ausgabe Schrittnummer
      #Schritt_Nummer := #S_DISPLAY;

   // sequencer 1
   INITIAL_STEP Step1:   // S1
      interlock C := NOT #A_NOT_HALT;
      // Warten auf Start
              R    #HM_belegt
   END_STEP
   TRANSITION Trans1 FROM Step1 TO Step2   // T1
      := #A_EIN AND NOT #HM_belegt;
   END_TRANSITION
   STEP Step4:   // S4
      interlock C := NOT #A_NOT_HALT;
      // Einfahrt bis Ende
      (C)     N    #Aggregat
   END_STEP
   TRANSITION Trans4 FROM Step4 TO Step5   // T4
      := #Sensor_Ende;
   END_TRANSITION
   STEP Step5:   // S5
      interlock C := NOT #A_NOT_HALT;
      // Warten auf Ausfahrt
   END_STEP
   TRANSITION Trans5 FROM Step5 TO Step6   // T5
      := #Nachfolgendes_Agg_frei AND #Sensor_Ende AND #A_EIN;
   END_TRANSITION
   STEP Step6:   // S6
      interlock C := NOT #A_NOT_HALT;
      // Ausfahrt bis Ende
      (C)     N    #Aggregat
   END_STEP
   TRANSITION Trans6 FROM Step6 TO Step1   // T6, jump
      := (#Step6.T > t#1s) AND NOT #Sensor_Ende;
   END_TRANSITION
   STEP Step3:   // S3
      interlock C := NOT #A_NOT_HALT;
      // Einfahrt Start
      (C)     N    #Aggregat
              S    #HM_belegt
   END_STEP
   TRANSITION Trans3 FROM Step3 TO Step4   // T3
      := #Step3.T > T#100MS;
   END_TRANSITION
   STEP Step2:   // S2
   END_STEP
   TRANSITION Trans2 FROM Step2 TO Step3   // T2
      := #A_EIN AND #Sensor_vorheriges_Agg AND NOT #HM_belegt;
   END_TRANSITION
END_FUNCTION_BLOCK

// ===== library: MasterCopy "Baustein_1" =====

FUNCTION_BLOCK "Baustein_1"   // FB2222, GRAPH
{ S7_Optimized_Access := 'FALSE' }
VERSION : 0.1
   VAR_INPUT
      INIT_SQ : Bool := false;   // Kette in Initialzustand versetzen
      A_EIN : Bool;
      A_NOT_HALT : Bool;
      Nachfolgendes_Agg_frei : Bool;
      Sensor_vorheriges_Agg : Bool;
      Sensor_Anfang : Bool;   // Öffner
      Sensor_Ende : Bool;   // Öffner
   END_VAR
   VAR_OUTPUT
      Schritt_Nummer : Int;
      Aggregat : Bool;
      Aggregat_frei : Bool;
   END_VAR
   VAR
      HM_FLAM : Array[1..8] of Bool;
      Flanke : Array[1..8] of Bool;
      HM_Agg_Frei : Bool;
      HM_belegt : Bool;
      SWITCH : Array[0..0] of DWord;
      SW_SQTS : Array[0..6] of Byte;
      SW_ADDR : Word := 16#C;
      G7T_0 : GraphTransition;
      G7S_0 : GraphStep;
      PRE_CRIT : Array[0..1] of DWord;
      POST_CRIT : Array[0..0] of DWord;
      TVX : Array[0..2] of Byte;
      TTX : Array[0..2] of Byte;
      TSX : Array[0..2] of Byte;
      S00X : Array[0..2] of Byte;
      SOFFX : Array[0..2] of Byte;
      SONX : Array[0..2] of Byte;
      SAX : Array[0..2] of Byte;
      SERRX : Array[0..7] of Byte;
      SMX : Array[0..7] of Byte;
      S0X : Array[0..7] of Byte;
      S1X : Array[0..7] of Byte;
      S_DISPLAY : Int;   // Interne Anzeige des Ausgangsparameters S_NO
      S_SEL_OLD : Int;   // Vorheriger Wert an S_SEL
      S_DISPIDX : Byte;   // Index des Schritts, der an S_NO anliegt
      T_DISPIDX : Byte;   // Index der Transition, die an T_NO anliegt
      MOPEDGE : Struct
         AUTO : Bool := false;
         MAN : Bool := false;
         TAP : Bool := false;
         TOP : Bool := false;
         ACK_S : Bool := false;
         REG_S : Bool := false;
         T_PREV : Bool := false;
         T_NEXT : Bool := false;
         LOCK : Bool := false;
         SUP : Bool := false;
         ACKREQ : Bool := false;
         SSKIP : Bool := false;
         OFF : Bool := false;
         INIT : Bool := false;
         HALT : Bool := false;
         TMS_HALT : Bool := false;
         OPS_ZERO : Bool := false;
         SACT_DISP : Bool := false;
         SEF_DISP : Bool := false;
         SALL_DISP : Bool := false;
         S_PREV : Bool := false;
         S_NEXT : Bool := false;
         S_SELOK : Bool := false;
         S_ON : Bool := false;
         S_OFF : Bool := false;
         T_PUSH : Bool := false;
         REG : Bool := false;
         ACK : Bool := false;
         IL_PERM : Bool := false;
         T_PERM : Bool := false;
         ILP_MAN : Bool := false;
      END_STRUCT;
      MOP : Struct   // Betriebsart
         AUTO : Bool := true;   // Zustand: Automatischer Betrieb
         MAN : Bool := false;   // Zustand: Handbetrieb
         TAP : Bool := false;   // Zustand: Halbautomatisch/Weiterschalten mit Transition
         TOP : Bool := false;   // Zustand: Halbautomatisch/Ignoriere Transition
         ACK_S : Bool := false;   // Anforderung: Schritt quittieren, der an Parameter S_NO anliegt
         REG_S : Bool := false;   // Anforderung: Schritt registrieren, der an Parameter S_NO anliegt
         T_PREV : Bool := false;   // Anforderung: Vorherige gültige Transition am Parameter T_NO ausgeben
         T_NEXT : Bool := false;   // Anforderung: Nächste gültige Transition am Parameter T_NO ausgeben
         LOCK : Bool := true;   // Zustand: Interlockbearbeitung aktiviert
         SUP : Bool := true;   // Zustand: Supervisionsbearbeitung aktiviert
         ACKREQ : Bool := false;   // Zustand: Quittierung erforderlich
         SSKIP : Bool := false;   // Zustand: "Schritte überspringen" aktiviert
         OFF : Bool := false;   // Anforderung: Alle Schritte deaktivieren
         INIT : Bool := true;   // Anforderung: Kette in Initialzustand schalten
         HALT : Bool := false;   // Zustand: Kette schaltet nicht weiter
         TMS_HALT : Bool := false;   // Zustand: Alle internen Zeiten angehalten
         OPS_ZERO : Bool := false;   // Zustand: Alle mit N, L, D bearbeitete Operanden auf 0 gesetzt
         SACT_DISP : Bool := true;   // Zustand: Nur aktive Schritte anzeigen
         SEF_DISP : Bool := false;   // Zustand: Nur fehlerhafte und gestörte Schritte anzeigen
         SALL_DISP : Bool := false;   // Zustand: Alle Schritte anzeigen
         S_PREV : Bool := false;   // Anforderung: Vorherigen Schritt am Parameter S_NO ausgeben
         S_NEXT : Bool := false;   // Anforderung: Nächsten Schritt am Parameter S_NO ausgeben
         S_SELOK : Bool := false;   // Anforderung: Schrittnummer, die am Parameter S_SEL anliegt, am Parameter S_NO ausgeben
         S_ON : Bool := false;   // Anforderung: Schritt aktivieren, der am Parameter S_NO anliegt
         S_OFF : Bool := false;   // Anforderung: Schritt deaktivieren, der am Parameter S_NO anliegt
         T_PUSH : Bool := false;   // Anforderung: Schaltfreigabe für Transition
         REG : Bool := false;   // Anforderung: Alle Interlock- und Supervisionsfehler registrieren
         ACK : Bool := false;   // Anforderung: Alle Interlock- und Supervisionsfehler quittieren
         IL_PERM : Bool := false;   // Zustand: Permanente Bearbeitung aller Interlocks
         T_PERM : Bool := false;   // Zustand: Permanente Bearbeitung aller Transitionen
         ILP_MAN : Bool := false;   // Zustand: Permanente Bearbeitung aller Interlocks im Handbetrieb
      END_STRUCT;
      TICKS : Struct   // Zeittakte
         DELTA : Time := T#0ms;   // Zeitdifferenz zwischen zwei Zyklen
         OLD : Time := T#0ms;   // 10 ms Taktzählerstand im letzten Zyklus
         NEW : Time := T#0ms;   // 10 ms Taktzählerstand in diesem Zyklus
      END_STRUCT;
      SQ_FLAGS : Struct   // Kettenmerker
         ERR_FLT : Bool := false;   // Sammelfehler Interlock und Supervision
         ERROR : Bool := false;   // Sammelfehler Interlock
         FAULT : Bool := false;   // Sammelfehler Supervision
         RT_FAIL : Bool := false;   // Laufzeitfehler
         NO_SNO : Bool := false;   // Angeforderte Schrittnummer nicht gefunden
         NF_OFL : Bool := false;   // Überlauf: Zu viele Anforderungen ON oder OFF
         SA_OFL : Bool := false;   // Überlauf: Zu viele Schritte aktiv
         TV_OFL : Bool := false;   // Überlauf: Zu viele gültige Transitionen
         MSG_OFL : Bool := false;   // Überlauf: Nicht genügend Systemressourcen fü ALARM_S
         NO_SWI : Bool := false;   // Nicht Schalten in diesem Zyklus
         CYC_OP : Bool := false;   // Zyklische Bearbeitung der Kette nach Initialisierung
         AS_MSG : Bool := true;   // Meldungen zur Laufzeit durch Anweisung aktiviert oder deaktiviert
         AS_SEND : Bool := false;   // Meldungen von WR_USMSG senden oder nur in Diagnosepuffer eintragen
         SQ_BUSY : Bool := false;   // Interner Flankenmerker für Vorgangsbearbeitung
         SA_BUSY : Bool := false;   // Interner Flankenmerker für Vorgangsbearbeitung
         AS_SIG : Bool := false;   // Flankenmerker für Meldungen von Alarm_S und Alarm_SQ
      END_STRUCT;
      S_PTR : DWord := 16#450;
      S_PTR2 : DWord := 16#0;
      S_PTR3 : DWord := 16#D50;
      S_PTR4 : DWord := 16#D10;
      T_PTR : DWord := 16#CD0;
      C_AR2 : DWord := 16#0;
      M_FBDB : DWord := 16#8AE0000;
      M_SNO : Word := 16#4;
      M_EVID : Word := 16#0;
      M_EVIL : C_Alarm_s;
      M_EVSV : C_Alarm_s;
      M_EV : DWord := 16#C30;
      CRIT : Array[0..31] of Bool;
      S_START : Byte := 16#0;
      S_IDX : Byte := 16#0;
      S_INT : Int := 72;
      S_TMP : Byte := 16#0;
      T_START : Byte := 16#0;
      T_IDX : Byte := 16#0;
      T_TMP : Byte := 16#0;
      T_TMP2 : Byte := 16#00;
      TV_POT : Byte := 16#02;
      RETURN1 : Byte := 16#0;
      RETURN2 : Byte := 16#0;
      SINI : Array[0..2] of Byte;
      LSTT : Array[0..6] of Byte;
      ATAJ : Array[0..6] of Byte;
      ATAB : Array[0..6] of Byte;
      PSTT : Array[0..6] of Byte;
      NSTT : Array[0..6] of Byte;
      ASSJ : Array[0..6] of Byte;
      ASSB : Array[0..6] of Byte;
      PTTS : Array[0..6] of Byte;
      NTTS : Array[0..6] of Byte;
      PRE_CNT : Word := 16#2;
      POST_CNT : Word := 16#1;
      ADR_COND : Word := 16#0;
      MAX_TVAL : Byte := 16#1;
      MAX_SACT : Byte := 16#1;
      MAX_CRIT : Byte := 16#4;
      T_CNT : Byte := 16#6;
      SUP_CNT : Byte := 16#0;
      LOCK_CNT : Byte := 16#5;
      S_CNT : Byte := 16#6;
      SQ_CNT : Byte := 16#1;
      PRS_INPAR : DWord := 16#40000000;
      PRS_OUTPAR : DWord := 16#0;
      GC_FLAGS : Struct
         T_MACH : Byte := 16#EB;
         COND_ED : Byte := 16#E2;
         W_LEVEL : Byte := 16#D5;
         FB_IF : Byte := 16#FA;
         AS_MSG : Word := 16#404;
         SSB : Word := 16#108;
         DILG : Word := 16#27E;
         ADDR_T0 : Word := 16#1A;
         CRIT_AVAIL : Bool := false;
         SSKIP_AVAIL : Bool := true;
         SSKIP_ON : Bool := false;
         ACK_REQ : Bool := false;
         SYNC_AVAIL : Bool := true;
         ILP_MAN : Bool := false;
         SWM_LOCKED : Bool := false;
         SAVE_SW : Bool := true;
      END_STRUCT;
      G7_FBMARK : Byte := 16#3C;
      G7_RELEASE : Byte := 16#3C;
      G7_ID2 : Byte := 16#37;
      G7_ID1 : Byte := 16#47;
   END_VAR
   // SW_SQTS[0] := 16#1;
   // TVX[0] := 16#1;
   // TTX[0] := 16#1;
   // TSX[0] := 16#1;
   // S00X[0] := 16#1;
   // SOFFX[0] := 16#1;
   // SONX[0] := 16#1;
   // SAX[0] := 16#1;
   // SERRX[0] := 16#1;
   // SMX[0] := 16#1;
   // S0X[0] := 16#1;
   // S1X[0] := 16#1;
   // SINI[0] := 16#2;
   // SINI[1] := 16#1;
   // SINI[2] := 0;
   // LSTT[0] := 0;
   // LSTT[1] := 0;
   // LSTT[2] := 0;
   // LSTT[3] := 0;
   // LSTT[4] := 0;
   // LSTT[5] := 0;
   // LSTT[6] := 16#1;
   // ATAJ[0] := 0;
   // ATAJ[1] := 16#1;
   // ATAJ[2] := 16#2;
   // ATAJ[3] := 16#3;
   // ATAJ[4] := 16#4;
   // ATAJ[5] := 16#5;
   // ATAJ[6] := 16#6;
   // ATAB[0] := 0;
   // ATAB[1] := 16#1;
   // ATAB[2] := 16#2;
   // ATAB[3] := 16#3;
   // ATAB[4] := 16#4;
   // ATAB[5] := 16#5;
   // ATAB[6] := 16#6;
   // PSTT[0] := 0;
   // PSTT[1] := 16#1;
   // PSTT[2] := 16#2;
   // PSTT[3] := 16#3;
   // PSTT[4] := 16#4;
   // PSTT[5] := 16#5;
   // PSTT[6] := 16#6;
   // NSTT[0] := 16#1;
   // NSTT[1] := 16#2;
   // NSTT[2] := 16#3;
   // NSTT[3] := 16#4;
   // NSTT[4] := 16#5;
   // NSTT[5] := 16#6;
   // NSTT[6] := 16#1;
   // ASSJ[0] := 0;
   // ASSJ[1] := 16#1;
   // ASSJ[2] := 16#2;
   // ASSJ[3] := 16#3;
   // ASSJ[4] := 16#4;
   // ASSJ[5] := 16#5;
   // ASSJ[6] := 16#6;
   // ASSB[0] := 0;
   // ASSB[1] := 16#1;
   // ASSB[2] := 16#2;
   // ASSB[3] := 16#3;
   // ASSB[4] := 16#4;
   // ASSB[5] := 16#5;
   // ASSB[6] := 16#6;
   // PTTS[0] := 0;
   // PTTS[2] := 16#1;
   // PTTS[3] := 16#2;
   // PTTS[4] := 16#3;
   // PTTS[5] := 16#4;
   // PTTS[6] := 16#5;
   // NTTS[0] := 0;
   // NTTS[1] := 16#1;
   // NTTS[2] := 16#2;
   // NTTS[3] := 16#3;
   // NTTS[4] := 16#4;
   // NTTS[5] := 16#5;
   // NTTS[6] := 16#6;
BEGIN
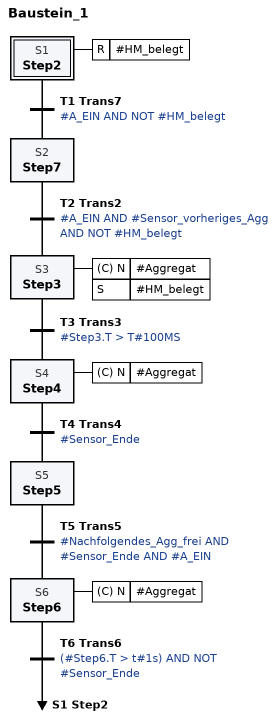
   // permanent pre-instructions
   NETWORK 1
      #HM_Agg_Frei := NOT #HM_belegt;
      #Aggregat_frei := NOT #HM_belegt;
   NETWORK 2
   TITLE = Ausgabe Schrittnummer
      #Schritt_Nummer := #S_DISPLAY;

   // sequencer 1
   INITIAL_STEP Step2:   // S1
      interlock C := NOT #A_NOT_HALT;
      // Warten auf Start
              R    #HM_belegt
   END_STEP
   TRANSITION Trans7 FROM Step2 TO Step7   // T1
      := #A_EIN AND NOT #HM_belegt;
   END_TRANSITION
   STEP Step4:   // S4
      interlock C := NOT #A_NOT_HALT;
      // Einfahrt bis Ende
      (C)     N    #Aggregat
   END_STEP
   TRANSITION Trans4 FROM Step4 TO Step5   // T4
      := #Sensor_Ende;
   END_TRANSITION
   STEP Step5:   // S5
      interlock C := NOT #A_NOT_HALT;
      // Warten auf Ausfahrt
   END_STEP
   TRANSITION Trans5 FROM Step5 TO Step6   // T5
      := #Nachfolgendes_Agg_frei AND #Sensor_Ende AND #A_EIN;
   END_TRANSITION
   STEP Step6:   // S6
      interlock C := NOT #A_NOT_HALT;
      // Ausfahrt bis Ende
      (C)     N    #Aggregat
   END_STEP
   TRANSITION Trans6 FROM Step6 TO Step2   // T6, jump
      := (#Step6.T > t#1s) AND NOT #Sensor_Ende;
   END_TRANSITION
   STEP Step3:   // S3
      interlock C := NOT #A_NOT_HALT;
      // Einfahrt Start
      (C)     N    #Aggregat
              S    #HM_belegt
   END_STEP
   TRANSITION Trans3 FROM Step3 TO Step4   // T3
      := #Step3.T > T#100MS;
   END_TRANSITION
   STEP Step7:   // S2
   END_STEP
   TRANSITION Trans2 FROM Step7 TO Step3   // T2
      := #A_EIN AND #Sensor_vorheriges_Agg AND NOT #HM_belegt;
   END_TRANSITION
END_FUNCTION_BLOCK